# B&R Automation Studio project Kontrol
Automation Studio 4.9

## Configuration Config1

CPU X20CP1382, AutomationRuntime D4.83, Build 4.1.2

### Task classes (Cpu.sw)
```
Cyclic#1 (cycle 2000 us, tolerance 2000 us):
  TaskFast <- Kontrol.TaskFast.TaskFast.prg
  FastMeter <- (binary)
  Program <- (binary)
  SslClient <- (binary)
  Server <- (binary)
  Client <- (binary)
  TEXC <- (binary)
  Modbus <- (binary)
Cyclic#2 (cycle 10000 us, tolerance 10000 us):
  Protection <- Kontrol.Protection.Protection.prg
  Control <- Kontrol.Control.Control.prg
Cyclic#3 (cycle 100000 us, tolerance 100000 us):
  WatchDog <- WatchDog.WatchDog.prg
  System <- Kontrol.System.System.prg
  Hardware <- Kontrol.Hardware.Hardware.prg
  ProtUpdate <- Kontrol.Protection.ProtUpdate.prg
  Command <- Kontrol.Command.Command.prg
  cb52 <- Kontrol.CB52.cb52.prg
Cyclic#4 (cycle 200000 us, tolerance 200000 us):
  Auto <- Auto.Auto.prg
  RV <- (binary)
  UHLM <- (binary)
  UHLM_AL <- (binary)
  Alarme <- (binary)
  DJ52G_IO <- (binary)
  Comandos <- (binary)
  RT <- (binary)
  SFA_IO <- (binary)
  FREIO <- (binary)
  UHRV_IO <- (binary)
  Comp_IO <- (binary)
  SC <- (binary)
  Comp_UH_AL <- (binary)
  Turbina_IO <- (binary)
  DJ52G <- (binary)
  UHRV <- (binary)
  SA <- (binary)
  Comp_UH_IO <- (binary)
  Gerador_AL <- (binary)
  Turbina_AL <- (binary)
  Comp_UH <- (binary)
  UHRV_AL <- (binary)
  Partida <- (binary)
  SFA <- (binary)
  UHLM_IO <- (binary)
  Gerador_IO <- (binary)
  Parada <- (binary)
  Status <- (binary)
  Comp <- (binary)
  Painel <- (binary)
  Energia <- (binary)
  FA <- (binary)
  Comp_AL <- (binary)
  SFA_AL <- (binary)
Cyclic#5 (cycle 500000 us, tolerance 500000 us):
  Nivel_IO <- (binary)
  Nivel <- (binary)
Cyclic#6 (cycle 100000 us, tolerance 3000000 us):
  MDB_Comand <- Auto.Modbus.MDB_Comando.prg
  MDB_Status <- Auto.Modbus.MDB_Status.prg
  MDB_Alarme <- Auto.Modbus.MDB_Alarme.prg
  MDB_Medida <- Auto.Modbus.MDB_Medida.prg
  MDB_Parame <- Auto.Modbus.MDB_Parametro.prg
Cyclic#7 (cycle 20000 us, tolerance 10000000 us):
  Event <- Kontrol.Event.Event.prg
  Comm <- Comm.Comm.prg
Cyclic#8 (cycle 50000 us, tolerance 10000000 us):
  File <- Kontrol.File.File.prg
Binaries: TCData, udbdef, ashwd, sysconf, asfw, arconfig, iomap, Role, User, ashwac, OpcUaMap, vccddbox, ihm01, ihm02, ihm03, vccpopup, vcpfx20, vcctrend, vccstr, vcmgr, vcpdsw, vcpdvnc, vccline, vccovl, arial, vcdsint, vccnum, vcalarm, vctcal, vccbtn, vcnet, vccbmp, vcrt, vcshared, vccdt, vcgclass, vcfntttf, vcbclass, vcdsloc, vcfile, arialbd, vcctext, vccshape, vccgauge, vcpkat, 10111548$f, Visu02, Visu03, Visu01, vccbar, vccslider, vcchspot, vccurl, vccalarm, vcchtml, vcxml
Libraries: operator, runtime, LoopConR, sys_lib, brsystem, AsTCP, AsIecCon, astime, AsBrStr, AsARCfg, AsXml, FileIO, AsIOAcc, standard, AsSem, IecCheck, DRV_mbus, dvframe, DataObj, Pgs0985, PgsAI4622, PgsAO4622, PgsAuto, PgsCfgNet, PgsComm, PgsControl, PgsEvent, PgsFileSys, PgsProt, PgsTag, PgsTagLink, PgsTelnet, vcresman, ashw
```

### Hardware
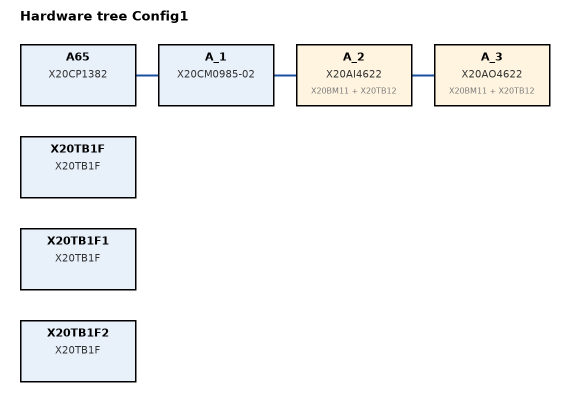
```
A65 : X20CP1382 v1.8.0.0  [X1 -> X1.SL; X2 -> X2.SL; X3 -> X3.SL]
  Module X1 (Type=X1, Virtual=true, Version=1.8.0.0)
    Connection (Connector=SS1, TargetModule=X20TB1F, TargetConnector=SS)
    Connection (Connector=SL, TargetModule=A65, TargetConnector=X1)
    X1AI_ChannelType01 = PT1000
    X1AI_ChannelType02 = 4 to 20mA
    X1AI2_LowerLimit_420mA = -8192
  Module X2 (Type=X2, Virtual=true, Version=1.8.0.0)
    Connection (Connector=SS1, TargetModule=X20TB1F1, TargetConnector=SS)
    Connection (Connector=SL, TargetModule=A65, TargetConnector=X2)
    X2CounterFunction = Edge
    X2CounterTimeInfo = 32Bit
  Module X3 (Type=X3, Virtual=true, Version=1.8.0.0)
    Connection (Connector=SS1, TargetModule=X20TB1F2, TargetConnector=SS)
    Connection (Connector=SL, TargetModule=A65, TargetConnector=X3)
  Connector IF2:
    ActivateDevice = 1
    HostName = kontrol
    Mode = Manual
    InternetAddress = 10.201.3.9
    SubnetMask = 255.255.255.192
    InaNodeNumber = 6
    Vnc1
    VncKeyMappingFile1 = 
    VncRefreshRate1 = 250
    ActivateSnmp = 2
    ActivateModbus = 1
    NumSlaves = -1
    NumAllBlocks = -1
    MemSizeIn = -1
    MemSizeOut = -1
  Connector IF3:
    CycleTime = 2000
    EPL_LossFrameTolerance_Selector = 2
    EPL_LossFrameTolerance = 5
    ActivateIna = 1
    InaNodeNumber = 1
  ConfigurationID = A65
  RemanentGlobalPvSize = 10940
  EnableUsbRemoteInstall = 1
  EnableCfRemoteInstall = 1
  SystemTick = 1000
  IdleTaskClass = 8
  TaskClassIdleTime = 4000
  Cyclic1Duration = 2000
  Cyclic1Tolerance = 2000
  Cyclic2Duration = 10000
  Cyclic2Tolerance = 10000
  Cyclic3Duration = 100000
  Cyclic3Tolerance = 100000
  Cyclic4Duration = 200000
  Cyclic4Tolerance = 200000
  Cyclic5Duration = 500000
  Cyclic5Tolerance = 500000
  Cyclic6Duration = 100000
  Cyclic6Tolerance = 3000000
  Cyclic7Duration = 20000
  Cyclic7Tolerance = 10000000
  Cyclic8Duration = 50000
  Cyclic8Tolerance = 10000000
  FileDevice1
  FileDeviceName1 = 
  FileDevicePath1 = 
  TimeZone = 105
  ActivateSntp = 1
  SntpcServAddr1 = a.st1.ntp.br
  SntpcServAddr2 = b.st1.ntp.br
  SntpcServAddr3 = c.st1.ntp.br
  SntpcServAddr4 = d.st1.ntp.br
  EthernetHostName = kontrol
  EthernetDefaultGateway = 10.201.3.62
  FtpUser1
  FtpUsername1 = progressul
  FtpUserPassword1 = vk2iY3J4UkERtYbEJrmZIzULlFJLyE0YoKo7iPp2s1I=
  FtpUserSalt1 = 6vig95Eg
  FTPAccessRight1 = 0
  FTPMSPartition1 = SYSTEM
  FTPMSpath1 = 
  ActivateOpcUa = 1
  OpcUaInformationModels_PV_Version = 1
A_1 : X20CM0985-02 v1.3.0.0  [X2X1 -> A65.IF6]
  Supervision = off
  ReadBack = on
  FuncDO5 = NetErrorUser
  Timestamps = on
  GenErrorReset = on
  GenErrorCheck = phaseline
  NetConfig = 3Phase
  SyncConfig = X4X3
A_2 : X20AI4622 v1.0.5.0  [SS1 -> X20TB12e.SS; SL -> X20BM11e.SL1]
  Supervision = off
  ChannelType01 = 4 to 20mA
  ChannelType02 = 4 to 20mA
  ChannelType03 = 4 to 20mA
  ChannelType04 = 4 to 20mA
A_3 : X20AO4622 v1.3.0.0  [SS1 -> X20TB12j.SS; SL -> X20BM11i.SL1]
  Supervision = off
  ChannelType01 = 0 to 20mA
  ChannelType02 = 4 to 20mA
  ChannelType03 = 4 to 20mA
  ChannelType04 = 4 to 20mA
X20BM11e : X20BM11 v1.0.0.1  [X2X1 -> A_1.X2X2]
X20BM11i : X20BM11 v1.0.0.1  [X2X1 -> X20BM11e.X2X2]
X20TB12e : X20TB12 v1.0.0.0
X20TB12j : X20TB12 v1.0.0.0
X20TB1F : X20TB1F v1.0.0.0
X20TB1F1 : X20TB1F v1.0.0.0
X20TB1F2 : X20TB1F v1.0.0.0
```

### IoMap.iom - A65/IoMap.iom
```iecst
(*********************************************************************************
 * Copyright: Microsoft
 * Author:    sandrionir
 * Created:   February 21, 2017/7:19 AM
 *********************************************************************************
 * IO mapping
 *********************************************************************************)
VAR_CONFIG
	Cyclic#2.::Control:rpm2.MasterCount AT %ID."X2".Counter02Value;
	Cyclic#2.::Control:rpm2.MasterTime AT %ID."X2".Counter02TimeChanged;
	Cyclic#2.::Control:rpm1.MasterCount AT %ID."X2".Counter01Value;
	Cyclic#2.::Control:rpm1.MasterTime AT %ID."X2".Counter01TimeChanged;
	Cyclic#2.cm0985IO.di.T32N AT %IX."A_1".StatusInput32;
	Cyclic#2.cm0985IO.di.T32P AT %IX."A_1".StatusInput31;
	Cyclic#2.cm0985IO.di.T27_2 AT %IX."A_1".StatusInput18;
	Cyclic#2.cm0985IO.di.T32Q AT %IX."A_1".StatusInput10;
	Cyclic#2.cm0985IO.di.T51 AT %IX."A_1".StatusInput09;
	Cyclic#2.cm0985IO.di.T50 AT %IX."A_1".StatusInput08;
	Cyclic#2.cm0985IO.di.T50N AT %IX."A_1".StatusInput07;
	Cyclic#2.cm0985IO.di.T60I AT %IX."A_1".StatusInput06;
	Cyclic#2.cm0985IO.di.T60V AT %IX."A_1".StatusInput05;
	Cyclic#2.cm0985IO.di.T81U AT %IX."A_1".StatusInput04;
	Cyclic#2.cm0985IO.di.T81O AT %IX."A_1".StatusInput03;
	Cyclic#2.cm0985IO.di.T27_1 AT %IX."A_1".StatusInput02;
	Cyclic#2.cm0985IO.di.T59 AT %IX."A_1".StatusInput01;
	Cyclic#2.cm0985IO.di.UgPhSeqFault AT %IX."A_1".StatusInput19;
	Cyclic#2.cm0985IO.di.IgPhSeqFault AT %IX."A_1".StatusInput20;
	Cyclic#2.cm0985IO.di.UbPhSeqFault AT %IX."A_1".StatusInput21;
	Cyclic#2.cm0985IO.di.Us1PhSeqFault AT %IX."A_1".StatusInput22;
	Cyclic#2.cm0985IO.di.PS24VFault AT %IX."A_1".StatusInput16;
	Cyclic#2.cm0985IO.do.RstError AT %QX."A_1".ResetGeneratorErrors;
	Cyclic#2.cm0985IO.do.INVDO05 AT %QX."A_1".InvertDO5;
	Cyclic#2.cm0985IO.do.SyncDeadBus AT %QX."A_1".ConfigOutput19;
	Cyclic#2.cm0985IO.do.SyncCheck AT %QX."A_1".ConfigOutput18;
	Cyclic#2.cm0985IO.do.SyncSlip AT %QX."A_1".ConfigOutput17;
	Cyclic#2.cm0985Meter.Registers.AnalogInput43 AT %ID."A_1".AnalogInput43;
	Cyclic#2.cm0985Meter.Registers.AnalogInput42 AT %ID."A_1".AnalogInput42;
	Cyclic#2.cm0985Meter.Registers.AnalogInput41 AT %ID."A_1".AnalogInput41;
	Cyclic#2.cm0985Meter.Registers.AnalogInput40 AT %ID."A_1".AnalogInput40;
	Cyclic#2.cm0985Meter.Registers.AnalogInput39 AT %ID."A_1".AnalogInput39;
	Cyclic#2.cm0985Meter.Registers.AnalogInput38 AT %ID."A_1".AnalogInput38;
	Cyclic#2.cm0985Meter.Registers.AnalogInput35 AT %IW."A_1".AnalogInput35;
	Cyclic#2.cm0985Meter.Registers.AnalogInput30 AT %IW."A_1".AnalogInput30;
	Cyclic#2.cm0985Meter.Registers.AnalogInput29 AT %IW."A_1".AnalogInput29;
	Cyclic#2.cm0985Meter.Registers.AnalogInput27 AT %IW."A_1".AnalogInput27;
	Cyclic#2.cm0985Meter.Registers.AnalogInput26 AT %IW."A_1".AnalogInput26;
	Cyclic#2.cm0985Meter.Registers.AnalogInput25 AT %IW."A_1".AnalogInput25;
	Cyclic#2.cm0985Meter.Registers.AnalogInput24 AT %IW."A_1".AnalogInput24;
	Cyclic#2.cm0985Meter.Registers.AnalogInput23 AT %IW."A_1".AnalogInput23;
	Cyclic#2.cm0985Meter.Registers.AnalogInput22 AT %IW."A_1".AnalogInput22;
	Cyclic#2.cm0985Meter.Registers.AnalogInput21 AT %IW."A_1".AnalogInput21;
	Cyclic#2.cm0985Meter.Registers.AnalogInput20 AT %IW."A_1".AnalogInput20;
	Cyclic#2.cm0985Meter.Registers.AnalogInput19 AT %IW."A_1".AnalogInput19;
	Cyclic#2.cm0985Meter.Registers.AnalogInput18 AT %IW."A_1".AnalogInput18;
	Cyclic#2.cm0985Meter.Registers.AnalogInput17 AT %IW."A_1".AnalogInput17;
	Cyclic#2.cm0985Meter.Registers.AnalogInput16 AT %IW."A_1".AnalogInput16;
	Cyclic#2.cm0985Meter.Registers.AnalogInput15 AT %IW."A_1".AnalogInput15;
	Cyclic#2.cm0985Meter.Registers.AnalogInput14 AT %IW."A_1".AnalogInput14;
	Cyclic#2.cm0985Meter.Registers.AnalogInput13 AT %IW."A_1".AnalogInput13;
	Cyclic#2.cm0985Meter.Registers.AnalogInput12 AT %IW."A_1".AnalogInput12;
	Cyclic#2.cm0985Meter.Registers.AnalogInput11 AT %IW."A_1".AnalogInput11;
	Cyclic#2.cm0985Meter.Registers.AnalogInput10 AT %IW."A_1".AnalogInput10;
	Cyclic#2.cm0985Meter.Registers.AnalogInput09 AT %IW."A_1".AnalogInput09;
	Cyclic#2.cm0985Meter.Registers.AnalogInput08 AT %IW."A_1".AnalogInput08;
	Cyclic#2.cm0985Meter.Registers.AnalogInput07 AT %IW."A_1".AnalogInput07;
	Cyclic#2.cm0985Meter.Registers.AnalogInput06 AT %IW."A_1".AnalogInput06;
	Cyclic#2.cm0985Meter.Registers.AnalogInput05 AT %IW."A_1".AnalogInput05;
	Cyclic#2.cm0985Meter.Registers.AnalogInput04 AT %IW."A_1".AnalogInput04;
	Cyclic#2.cm0985Meter.Registers.AnalogInput03 AT %IW."A_1".AnalogInput03;
	Cyclic#2.cm0985Meter.Registers.AnalogInput02 AT %IW."A_1".AnalogInput02;
	Cyclic#2.cm0985Meter.Registers.AnalogInput01 AT %IW."A_1".AnalogInput01;
	Cyclic#2.cm0985Meter.Registers.AnalogInput33 AT %IW."A_1".AnalogInput33;
	Cyclic#2.cm0985Meter.Registers.AnalogInput34 AT %IW."A_1".AnalogInput34;
	Cyclic#2.cm0985Meter.Registers.AnalogInput31 AT %IW."A_1".AnalogInput31;
	Cyclic#2.cm0985Meter.Registers.AnalogInput32 AT %IW."A_1".AnalogInput32;
	HW.SerialNumber AT %ID."A65".SerialNumber;
	HW.ModuleID AT %IW."A65".ModuleID;
	HW.TemperatureENV AT %IW."A65".TemperatureENV;
	HW.TemperatureCPU AT %IW."A65".TemperatureCPU;
	HW.FalhaFonteIO AT %IX."X3".StatusInput01;
	HW.Modulos.X1_Status AT %IB."X1".StatusInput01;
	HW.Modulos.A_1_OK AT %IX."A_1".ModuleOk;
	HW.Modulos.A_2_OK AT %IX."A_2".ModuleOk;
	HW.Modulos.A_3_OK AT %IX."A_3".ModuleOk;
	Protection.ai.ExcTemp AT %IW."X1".AnalogInput01;
	A65.ai.if AT %IW."X1".AnalogInput02;
	A65.ai.uf AT %IW."A_2".AnalogInput01;
	A65.ai.pos1 AT %IW."A_2".AnalogInput02;
	A65.ai.pos2 AT %IW."A_2".AnalogInput03;
	A65.ai.pos3 AT %IW."A_2".AnalogInput04;
	A65.ao.pwr AT %QW."A_3".AnalogOutput01;
	A65.ao.pos1 AT %QW."A_3".AnalogOutput02;
	A65.ao.pos2 AT %QW."A_3".AnalogOutput03;
	A65.ao.pos3 AT %QW."A_3".AnalogOutput04;
	A65.di.reset  AT %IX."X1".DigitalInput01;
	A65.di.gov_enable  AT %IX."X1".DigitalInput02;
	A65.di.gov_ctrl_pwr_enable AT %IX."X1".DigitalInput03;
	A65.di.gov_unload AT %IX."X1".DigitalInput04;
	A65.di.avr_enable AT %IX."X2".DigitalInput01;
	A65.di.avr_ctrl_qm_enable AT %IX."X2".DigitalInput02;
	A65.di.avr_ctrl_pf_enable AT %IX."X2".DigitalInput03;
	A65.di.sync_enable AT %IX."X2".DigitalInput04;
	A65.di.dead_bus_enable AT %IX."X2".DigitalInput05;
	A65.di.remote AT %IX."X2".DigitalInput07;
	A65.di.gov_trip AT %IX."X2".DigitalInput08;
	A65.di.avr_trip AT %IX."X2".DigitalInput09;
	CB52.di.closed AT %IX."X2".DigitalInput06;
	Protection.di.crowbar_ok AT %IX."X2".DigitalInput10;
	Protection.di.pwr_temp_ok AT %IX."X2".DigitalInput14;
	Protection.do.trip_86e AT %QX."A_1".DigitalOutput05;
	Protection.do.trip_86h AT %QX."A_1".DigitalOutput06;
	Protection.do.trip_50bf AT %QX."X3".DigitalOutput12;
	A65.do.gov_on AT %QX."X3".DigitalOutput02;
	A65.do.watchdog AT %QX."X3".DigitalOutput01;
	A65.do.power_zero AT %QX."X3".DigitalOutput03;
	A65.do.rotation_zero AT %QX."X3".DigitalOutput04;
	A65.do.rotation_nominal AT %QX."X3".DigitalOutput05;
	A65.do.rotation_brake AT %QX."X3".DigitalOutput06;
	A65.do.avr_on AT %QX."X3".DigitalOutput07;
	A65.do.field_flash_on AT %QX."X3".DigitalOutput08;
	A65.do.voltage_nominal AT %QX."X3".DigitalOutput09;
	A65.do.sync_enabled AT %QX."X3".DigitalOutput10;
	A65.do.dead_bus_enabled AT %QX."X3".DigitalOutput11;
END_VAR
```

## Logical view

Binary libraries used (declarations not repeated): operator, runtime, LoopConR 4.10.0, sys_lib, brsystem, AsTCP, AsIecCon, astime, AsARCfg, FileIO, standard, AsSem, AsIOAcc, AsXml, AsBrStr, DRV_mbus, dvframe, DataObj, IecCheck, Pgs0985, PgsAI4622 1.00.0, PgsAO4622 1.00.0, PgsCfgNet 2.02.0, PgsComm, PgsControl 2.03.3, PgsEvent, PgsFileSys 2.00.0, PgsTag, PgsTagLink 2.00.0, PgsTelnet

### Package Logical/Libraries - Global libraries

### Library Logical/Libraries/Kontrol/PgsAuto (IEC)
Depends on: sys_lib

#### Types.typ - Exported data types
```iecst
TYPE
	PgsHorimetroPrivType : 	STRUCT
		init : BOOL := TRUE;
		init_ton : TON;
		sec_old : USINT;
		rtc_time : RTCtime_typ;
		bkp_ton : TON;
	END_STRUCT;
	PgsManobraPrivType : 	STRUCT
		init : BOOL := TRUE;
		init_ton : TON;
		bkp_ton : TON;
		m : BOOL;
	END_STRUCT;
	PgsEnergiaPrivType : 	STRUCT
		init : BOOL := TRUE;
		init_ton : TON;
		dh : REAL; (*Delta Hour*)
		rt_info : RTInfo;
		bkp_ton : TON;
	END_STRUCT;
END_TYPE
```

#### PgsAuto.fun - Exported functions and function blocks
```iecst
FUNCTION_BLOCK PgsEnergia
	VAR_INPUT
		enable : BOOL;
		reset : BOOL;
		power : REAL;
		set_inicial : BOOL;
		set_posEnergy : REAL;
		set_negEnergy : REAL;
	END_VAR
	VAR_OUTPUT
		posEnergy : LREAL;
		negEnergy : LREAL;
	END_VAR
	VAR
		priv : PgsEnergiaPrivType;
	END_VAR
END_FUNCTION_BLOCK

FUNCTION_BLOCK PgsHorimetro
	VAR_INPUT
		enable : BOOL;
		reset : BOOL;
		set_inicial : BOOL;
		set_total : REAL;
	END_VAR
	VAR_OUTPUT
		total : REAL;
		horas : REAL;
		minutos : REAL;
		segundos : REAL;
	END_VAR
	VAR
		priv : PgsHorimetroPrivType;
	END_VAR
END_FUNCTION_BLOCK

FUNCTION_BLOCK PgsManobra
	VAR_INPUT
		enable : BOOL;
		reset : BOOL;
		set_inicial : BOOL;
		set_total : REAL;
	END_VAR
	VAR_OUTPUT
		total : REAL;
	END_VAR
	VAR
		priv : PgsManobraPrivType;
	END_VAR
END_FUNCTION_BLOCK

FUNCTION PGS_MDB_TO_REAL : REAL (*TODO: Add your comment here*) (*$GROUP=User,$CAT=User,$GROUPICON=User.png,$CATICON=User.png*)
	VAR_INPUT
		IN : UDINT;
	END_VAR
	VAR
		pVar : REFERENCE TO REAL;
		varUint : ARRAY[0..1] OF UINT;
		varUint1 : REFERENCE TO ARRAY[0..1] OF UINT;
	END_VAR
END_FUNCTION

FUNCTION PGS_REAL_TO_MDB : UDINT (*TODO: Add your comment here*) (*$GROUP=User,$CAT=User,$GROUPICON=User.png,$CATICON=User.png*)
	VAR_INPUT
		IN : REAL;
	END_VAR
	VAR
		pVar : REFERENCE TO UDINT;
		varUint : ARRAY[0..1] OF UINT;
		varUint1 : REFERENCE TO ARRAY[0..1] OF UINT;
	END_VAR
END_FUNCTION

{REDUND_ERROR} FUNCTION PGS_MDB_TO_DINT : DINT (*TODO: Add your comment here*) (*$GROUP=User,$CAT=User,$GROUPICON=User.png,$CATICON=User.png*)
	VAR_INPUT
		HIGH : UINT;
		LOW : UINT;
	END_VAR
	VAR
		pVar : REFERENCE TO DINT;
		varUint : ARRAY[0..1] OF UINT;
	END_VAR
END_FUNCTION

{REDUND_ERROR} FUNCTION PGS_MDB_TO_UDINT : UDINT (*TODO: Add your comment here*) (*$GROUP=User,$CAT=User,$GROUPICON=User.png,$CATICON=User.png*)
	VAR_INPUT
		HIGH : UINT;
		LOW : UINT;
	END_VAR
	VAR
		pVar : REFERENCE TO UDINT;
		varUint : ARRAY[0..1] OF UINT;
	END_VAR
END_FUNCTION

FUNCTION_BLOCK PgsAlarme
	VAR_INPUT
		IN : BOOL; (*input signal*)
		PT : TIME; (*delay time*)
		RESET : BOOL; (*resets output Q1*)
	END_VAR
	VAR_OUTPUT
		Q : BOOL; (*rising edge of the input signal is delayed by PT*)
	END_VAR
	VAR
		ton : TON;
	END_VAR
END_FUNCTION_BLOCK

{REDUND_ERROR} FUNCTION_BLOCK PgsFiltro (*TODO: Add your comment here*) (*$GROUP=User,$CAT=User,$GROUPICON=User.png,$CATICON=User.png*)
	VAR_INPUT
		IN : {REDUND_UNREPLICABLE} REAL;
		CTE : {REDUND_UNREPLICABLE} REAL;
	END_VAR
	VAR_OUTPUT
		OUT : {REDUND_UNREPLICABLE} REAL;
	END_VAR
	VAR
		acc : REAL;
	END_VAR
END_FUNCTION_BLOCK

{REDUND_ERROR} FUNCTION_BLOCK PgsEscala (*TODO: Add your comment here*) (*$GROUP=User,$CAT=User,$GROUPICON=User.png,$CATICON=User.png*)
	VAR_INPUT
		SensorMax : {REDUND_UNREPLICABLE} REAL;
		SensorMin : {REDUND_UNREPLICABLE} REAL;
		Filtro : REAL;
		Entrada : REAL;
	END_VAR
	VAR_OUTPUT
		Valor : {REDUND_UNREPLICABLE} REAL;
		Sensor : REAL;
	END_VAR
	VAR
		priv_filtro : PgsFiltro;
		priv_first_start : BOOL;
	END_VAR
END_FUNCTION_BLOCK

{REDUND_ERROR} FUNCTION_BLOCK PgsCabo (*TODO: Add your comment here*) (*$GROUP=User,$CAT=User,$GROUPICON=User.png,$CATICON=User.png*)
	VAR_INPUT
		IN : REAL;
		PT : TIME;
	END_VAR
	VAR_OUTPUT
		Falha : BOOL;
		Cabo_Aberto : BOOL;
		Cabo_Curto : BOOL;
	END_VAR
	VAR
		aberto : BOOL;
		curto : BOOL;
		ton_aberto : TON;
		ton_curto : TON;
	END_VAR
END_FUNCTION_BLOCK

{REDUND_OK} FUNCTION_BLOCK PgsSobre (*TODO: Add your comment here*) (*$GROUP=User,$CAT=User,$GROUPICON=User.png,$CATICON=User.png*)
	VAR_INPUT
		enable : BOOL := TRUE;
		IN : REAL;
		IN_AL : REAL;
		PT_AL : REAL;
		IN_TP : REAL;
		PT_TP : REAL;
		RST : BOOL;
	END_VAR
	VAR_OUTPUT
		Alarme : BOOL;
		Trip : BOOL;
	END_VAR
	VAR
		ton_al : TON;
		ton_tp : TON;
	END_VAR
END_FUNCTION_BLOCK

{REDUND_OK} FUNCTION_BLOCK PgsSub (*TODO: Add your comment here*) (*$GROUP=User,$CAT=User,$GROUPICON=User.png,$CATICON=User.png*)
	VAR_INPUT
		enable : BOOL := TRUE;
		IN : REAL;
		IN_AL : REAL;
		PT_AL : REAL;
		IN_TP : REAL;
		PT_TP : REAL;
		RST : BOOL;
	END_VAR
	VAR_OUTPUT
		Alarme : BOOL;
		Trip : BOOL;
	END_VAR
	VAR
		ton_al : TON;
		ton_tp : TON;
	END_VAR
END_FUNCTION_BLOCK

FUNCTION_BLOCK PgsX20AT
	VAR_INPUT
		Status : USINT;
	END_VAR
	VAR_OUTPUT
		IN1_Aberto : BOOL;
		IN1_Curto : BOOL;
		IN2_Aberto : BOOL;
		IN2_Curto : BOOL;
		IN3_Aberto : BOOL;
		IN3_Curto : BOOL;
		IN4_Aberto : BOOL;
		IN4_Curto : BOOL;
	END_VAR
END_FUNCTION_BLOCK

{REDUND_ERROR} FUNCTION_BLOCK PgsEscalaTotal (*TODO: Add your comment here*) (*$GROUP=User,$CAT=User,$GROUPICON=User.png,$CATICON=User.png*)
	VAR_INPUT
		SensorMax : {REDUND_UNREPLICABLE} REAL;
		SensorMin : {REDUND_UNREPLICABLE} REAL;
		ValorMax : {REDUND_UNREPLICABLE} REAL;
		ValorMin : {REDUND_UNREPLICABLE} REAL;
		Entrada : REAL;
	END_VAR
	VAR_OUTPUT
		Valor : {REDUND_UNREPLICABLE} REAL;
		Sensor : REAL;
	END_VAR
END_FUNCTION_BLOCK
```

#### PgsHorimetro.st
```iecst
FUNCTION_BLOCK PgsHorimetro

	priv.init_ton(IN:= priv.init, PT:=T#10s);
	IF priv.init_ton.Q THEN
		priv.init := FALSE;
		total := set_total;
	END_IF;

	RTC_gettime(ADR(priv.rtc_time));
	IF reset THEN
		reset 	:= FALSE;
		total 	:= 0.0;
	END_IF;

	IF enable AND priv.sec_old <> priv.rtc_time.second THEN
		total := total + 1.0 / 3600.0;
	END_IF;
	priv.sec_old := priv.rtc_time.second;

	IF set_inicial THEN
		set_inicial := FALSE;
		total := set_total;
	END_IF;

	horas	:= TRUNC(total);
	minutos	:= TRUNC((total - horas)*60.0);
	segundos:= TRUNC((total - horas - minutos/60.0)*3600.0);

	priv.bkp_ton(IN:= NOT priv.bkp_ton.Q, PT:=T#10m);
	IF priv.bkp_ton.Q THEN
		set_total := total;
	END_IF;
END_FUNCTION_BLOCK
```

#### PgsManobra.st
```iecst
FUNCTION_BLOCK PgsManobra
	priv.init_ton(IN:= priv.init, PT:=T#10s);
	IF priv.init_ton.Q THEN
		priv.init := FALSE;
		total := set_total;
	END_IF;

    IF reset THEN
    	reset	:= FALSE;
        total	:= 0;
    END_IF;

	IF set_inicial THEN
		set_inicial	:= FALSE;
		total	:= set_total;
	END_IF;

    IF NOT priv.m AND enable THEN total := total + 1.0; END_IF;
    priv.m := enable;

	priv.bkp_ton(IN:= NOT priv.bkp_ton.Q, PT:=T#1m);
	IF priv.bkp_ton.Q THEN
		set_total := total;
	END_IF;
END_FUNCTION_BLOCK
```

#### PGS_MDB_TO_UDINT.st
```iecst
(* TODO: Add your comment here *)
FUNCTION PGS_MDB_TO_UDINT
    varUint[0] := HIGH;
    varUint[1] := LOW;
    pVar ACCESS ADR(varUint);
    PGS_MDB_TO_UDINT := pVar;
END_FUNCTION
```

#### PgsCabo.st
```iecst
(* TODO: Add your comment here *)
FUNCTION_BLOCK PgsCabo
	curto 	:= IN >= 20.0;
	aberto	:= IN <= 3.0;
	ton_aberto(IN:=aberto,PT:=PT);
	ton_curto(IN:=curto,PT:=PT);
	Falha 		:= aberto OR curto;
	Cabo_Aberto	:= ton_aberto.Q;
	Cabo_Curto	:= ton_curto.Q;
END_FUNCTION_BLOCK
```

#### PgsSub.st
```iecst
(*<$Description$> TODO: Add your comment here </$Description$>*)
FUNCTION_BLOCK PgsSub

	(* Alarme *)
	IF IN_AL = 0 THEN
		Alarme	:= FALSE;
	ELSE
		ton_al( IN := IN <= IN_AL , PT := REAL_TO_TIME( PT_AL * 1000) );
		IF ton_al.Q AND enable THEN
			Alarme	:= TRUE;
		ELSIF RST THEN
			Alarme	:= FALSE;
		END_IF;
	END_IF;

	(*Trip*)
	IF IN_TP = 0 THEN
		Trip	:= FALSE;
	ELSE
		ton_tp( IN := IN <= IN_TP , PT := REAL_TO_TIME( PT_TP * 1000) );
		IF ton_tp.Q AND enable THEN
			Trip	:= TRUE;
		ELSIF RST THEN
			Trip	:= FALSE;
		END_IF;
 	END_IF;

END_FUNCTION_BLOCK
```

#### PgsX20AT.st
```iecst
(*<$Description$> TODO: Add your comment here </$Description$>*)
FUNCTION_BLOCK PgsX20AT
	IN1_Aberto		:= Status.0;
	IN1_Curto		:= (Status.1 = 1) AND (Status.0 = 0);

	IN2_Aberto		:= Status.2;
	IN2_Curto		:= (Status.3 = 1) AND (Status.2 = 0);

	IN3_Aberto		:= Status.4;
	IN3_Curto		:= (Status.5 = 1) AND (Status.4 = 0);

	IN4_Aberto		:= Status.6;
	IN4_Curto		:= (Status.7 = 1) AND (Status.6 = 0);

END_FUNCTION_BLOCK
```

#### PgsEscalaTotal.st
```iecst
(* TODO: Add your comment here *)
FUNCTION_BLOCK PgsEscalaTotal

	Sensor	:= (Entrada / 32767.0) * 16.0 + 4.0;
	IF (SensorMax - SensorMin) <> 0 THEN
		Valor   := ((Sensor - SensorMin) / (SensorMax - SensorMin))
				* (ValorMax - ValorMin)
				+  ValorMin;
	ELSE
		Valor   := 0.0;
	END_IF;

END_FUNCTION_BLOCK
```

#### PgsEscala.st
```iecst
(* TODO: Add your comment here *)
FUNCTION_BLOCK PgsEscala

	Sensor	:= (Entrada / 32767.0) * 16.0 + 4.0;

	IF Filtro < 1 THEN
		Filtro := 1;
	END_IF
	priv_filtro(IN:=Sensor, CTE:=Filtro);

	IF NOT priv_first_start THEN
		priv_first_start := TRUE;
		priv_filtro(IN:= (Sensor - (priv_filtro.acc / Filtro) ) * Filtro);
	END_IF;

	Valor   := ((priv_filtro.OUT - 4.0) / 16.0)
	* (SensorMax - SensorMin)
	+  SensorMin;

END_FUNCTION_BLOCK
```

### Share.var
```iecst
VAR
	WDOK : BOOL := TRUE;
	License : PgsLicense;
END_VAR
```

### Program Logical/WatchDog/WatchDog

#### Cyclic.st
```iecst
PROGRAM _CYCLIC
    License();
    ProtFlag.KeyInvalid			:= NOT License.Valid;
    ProtFlag.PwrSrcCpuIOFault	:= HW.FalhaFonteIO;
    ProtFlag.PwrSrcM1IOFault	:= cm0985IO.di.PS24VFault;

    IF  License.Valid
    AND	NOT ProtFlag.PwrSrcCpuIOFault	// Power Source CPU I/O Fault
    AND	NOT ProtFlag.PwrSrcM1IOFault	// Power Source Energy Module I/O Fault
    AND	HW.Modulos.A_1_OK
    AND	HW.Modulos.A_2_OK
	AND	HW.Modulos.A_3_OK
//	AND	HW.Modulos.A_4_OK
//	AND	HW.Modulos.A_5_OK
//	AND	HW.Modulos.A_6_OK
//	AND	HW.Modulos.A_7_OK
//	AND	HW.Modulos.A_8_OK
//	AND	HW.Modulos.A_9_OK
//	AND	HW.Modulos.A_10_OK
//	AND	HW.Modulos.A_11_OK
//	AND	HW.Modulos.A_12_OK
	THEN
        WDOK    := TRUE;
    ELSE
        WDOK    := FALSE;
    END_IF

    //WatchDog
    ProtFlag.WatchDog	:= NOT WDOK;
	A65.do.watchdog		:= WDOK;

END_PROGRAM
```

- Cyclic.st.bak (not shown)

### Program Logical/Comm/Comm (IEC)

#### Variables.var
```iecst
VAR
	mbusData : PgsMbDataOpen;
	mbusDevice : PgsMbDevice;
	mbusSetBlock : PgsMbSetBlock;
	mbusSetLink : PgsMbSetLink;
	mbusDataClose : PgsMbDataClose;
	mbusLinkClose : PgsMbLinkClose;
	mbusTcpOpen : PgsMbTcpOpen;
	mbusTcpUpdate : PgsMbTcpUpdate;
	mbusTcpClose : PgsMbTcpClose;
	telnetOpen : PgsTelnetOpen;
	telnetUpdate : PgsTelnetUpdate;
	telnetClose : PgsTelnetClose;
END_VAR
(*Reset COM*)
VAR
	ton_reset_Tcp : TON;
END_VAR
```

#### Cyclic.st
```iecst
PROGRAM _CYCLIC

    IF NOT PgsTagValid(TagManager.ident) THEN
        RETURN;
    END_IF

    mbusTcpUpdate   ( ident := mbusTcpOpen.ident );
    telnetUpdate(
        ident       := telnetOpen.ident,
        tagIdent    := TagManager.ident,
        evtIdent    := Event
    );

	ton_reset_Tcp(IN:= A65.di.reset, PT:= T#30s);
	IF ton_reset_Tcp.Q THEN
		mbusTcpUpdate.reset := TRUE;
	END_IF;

END_PROGRAM
```

#### Exit.st
```iecst
PROGRAM _EXIT

	mbusDataClose( dtaIdent := mbusData.dtaIdent );

	mbusLinkClose( lnkIdent := link_avr.Ident );
	mbusLinkClose( lnkIdent := link_gov.Ident );

	mbusLinkClose( lnkIdent := link_pos1.Ident );
	mbusLinkClose( lnkIdent := link_pos2.Ident );
	mbusLinkClose( lnkIdent := link_pos3.Ident );
	mbusLinkClose( lnkIdent := link_curve1.Ident );
	mbusLinkClose( lnkIdent := link_curve2.Ident );
	mbusLinkClose( lnkIdent := link_curve3.Ident );

	mbusLinkClose( lnkIdent := link_meter.Ident );

	mbusLinkClose( lnkIdent := link_system.Ident );
	mbusLinkClose( lnkIdent := link_sysIO.Ident );
	mbusLinkClose( lnkIdent := link_prot.Ident );

    mbusTcpClose( enable := TRUE, ident := mbusTcpOpen.ident );

    telnetClose( enable := TRUE, ident := telnetOpen.ident );

END_PROGRAM
```

#### Init.st
```iecst
PROGRAM _INIT

    mbusData( Devices := 1 );

	//Device 1
    mbusDevice(
        dtaIdent        := mbusData.dtaIdent,
        id              := 1,
		Links			:= 6,
		InputBlocks		:= 1,
        CoilBlocks      := 3
    );

    //AVR
	link_avr(
		CoilAddress		:= 4097,
		HoldingAddress	:= 5121,
		InputAddress	:= 7169,
        //GainUm          := 10.0,
        //GainIm          := 10.0,
        //GainSm          := 10.0,
        //GainUf          := 100.0,
        //GainIf          := 100.0,
		Float			:= TRUE,
		ModiconFormat	:= TRUE
	);
	mbusSetLink(
		devIdent	:= mbusDevice.devIdent,
		lnkIdent	:= link_avr.Ident
	);

    //GOV
	link_gov(
		CoilAddress		:= 8193,
		HoldingAddress	:= 9217,
		InputAddress	:= 11265,
        //GainUm          := 10.0,
        //GainSm          := 10.0,
		Float			:= TRUE,
		ModiconFormat	:= TRUE
	);
	mbusSetLink(
		devIdent	:= mbusDevice.devIdent,
		lnkIdent	:= link_gov.Ident
	);

	//POS1
	link_pos1(
		CoilAddress		:= 12289,
		HoldingAddress	:= 12545,
		InputAddress	:= 13569,
		Float			:= TRUE,
		ModiconFormat	:= TRUE
	);
	mbusSetLink(
		devIdent	:= mbusDevice.devIdent,
		lnkIdent	:= link_pos1.Ident
	);
	//Curve1
	link_curve1(
		HoldingAddress	:= 13825,
		InputAddress	:= 13953,
		Float			:= TRUE,
		ModiconFormat	:= TRUE
	);
	mbusSetLink(
		devIdent	:= mbusDevice.devIdent,
		lnkIdent	:= link_curve1.Ident
	);

	//POS2
	link_pos2(
		CoilAddress		:= 14337,
		HoldingAddress	:= 14593,
		InputAddress	:= 15617,
		Float			:= TRUE,
		ModiconFormat	:= TRUE
	);
	mbusSetLink(
		devIdent	:= mbusDevice.devIdent,
		lnkIdent	:= link_pos2.Ident
	);
	//Curve2
	link_curve2(
		HoldingAddress	:= 15873,
		InputAddress	:= 16001,
		Float			:= TRUE,
		ModiconFormat	:= TRUE
	);
	mbusSetLink(
		devIdent	:= mbusDevice.devIdent,
		lnkIdent	:= link_curve2.Ident
	);

	//POS3
	link_pos3(
		CoilAddress		:= 16385,
		HoldingAddress	:= 16641,
		InputAddress	:= 17665,
		Float			:= TRUE,
		ModiconFormat	:= TRUE
	);
	mbusSetLink(
		devIdent	:= mbusDevice.devIdent,
		lnkIdent	:= link_pos3.Ident
	);
	//Curve3
	link_curve3(
		HoldingAddress	:= 17921,
		InputAddress	:= 18049,
		Float			:= TRUE,
		ModiconFormat	:= TRUE
	);
	mbusSetLink(
		devIdent	:= mbusDevice.devIdent,
		lnkIdent	:= link_curve3.Ident
	);

    // MdbMeter
	link_meter(
        pBlock	        := ADR(MdbMeter),
        blockLen	    := SIZEOF(MdbMeter),
		Address			:= 2561,
		Holding			:= FALSE,
		//Gain			:= 10.0,
		Float			:= TRUE,
		ModiconFormat	:= TRUE
	);
	mbusSetLink(
		devIdent	:= mbusDevice.devIdent,
		lnkIdent	:= link_meter.Ident
	);

    // System Parameter
	link_system(
        pBlock	        := ADR(SysPar),
        blockLen	    := SIZEOF(SysPar),
		Address			:= 1025,
		Holding			:= TRUE,
		//Gain			:= 10,
		Float			:= TRUE,
		ModiconFormat	:= TRUE
	);
	mbusSetLink(
		devIdent	:= mbusDevice.devIdent,
		lnkIdent	:= link_system.Ident
	);
    //
    link_sysIO(
        pBlock	        := ADR(SysIOPar),
        blockLen	    := SIZEOF(SysIOPar),
		Address			:= 1255,
		Holding			:= TRUE,
		//Gain			:= 10,
		Float			:= TRUE,
		ModiconFormat	:= TRUE
	);
	mbusSetLink(
		devIdent	:= mbusDevice.devIdent,
		lnkIdent	:= link_sysIO.Ident
	);

    //SysUpdate
 	mbusSetBlock(
        devIdent    := mbusDevice.devIdent,
        BlockType   := PGS_MB_BLK_COIL,
        Address     := 1,
        pBlock      := ADR(SysUpdate),
        blockLen    := SIZEOF(SysUpdate)
    );

    //Protections
 	mbusSetBlock(
        devIdent    := mbusDevice.devIdent,
        BlockType   := PGS_MB_BLK_COIL,
        Address     := 40961,
        pBlock      := ADR(ProtFlag),
        blockLen    := SIZEOF(ProtFlag)
	);
	// Protections Parameter
	link_prot(
		pBlock	        := ADR(ProtPar),
		blockLen	    := SIZEOF(ProtPar),
		Address			:= 41985,
		Holding			:= TRUE,
		//Gain			:= 10,
		Float			:= TRUE,
		ModiconFormat	:= TRUE
	);
	mbusSetLink(
		devIdent	:= mbusDevice.devIdent,
		lnkIdent	:= link_prot.Ident
	);

    //Automação
    link_mdb_medidas(
		pBlock	        := ADR(MDB_Medidas),
		blockLen	    := SIZEOF(MDB_Medidas),
		Address			:= 19089, (*50001*)
		Holding			:= FALSE,
		//Gain			:= 10,
		Float			:= TRUE,
		ModiconFormat	:= TRUE
	);
	mbusSetLink(
		devIdent	:= mbusDevice.devIdent,
		lnkIdent	:= link_mdb_medidas.Ident
	);
    link_mdb_parametros(
		pBlock	        := ADR(MDB_Parametros),
		blockLen	    := SIZEOF(MDB_Parametros),
		Address			:= 21589, (*50257*)
		Holding			:= TRUE,
		//Gain			:= 10,
		Float			:= TRUE,
		ModiconFormat	:= TRUE
	);
	mbusSetLink(
		devIdent	:= mbusDevice.devIdent,
		lnkIdent	:= link_mdb_parametros.Ident
	);
	mbusSetBlock(
		devIdent    := mbusDevice.devIdent,
		BlockType   := PGS_MB_BLK_COIL,
		Address     := 21889,
		pBlock      := ADR(MDB_Alarmes),
		blockLen    := SIZEOF(MDB_Alarmes)
	);
	mbusSetBlock(
        devIdent    := mbusDevice.devIdent,
        BlockType   := PGS_MB_BLK_COIL,
        Address     := 17089, (*50001*)
        pBlock      := ADR(MDB_Status),
        blockLen    := SIZEOF(MDB_Status)
    );
     mbusSetBlock(
        devIdent    := mbusDevice.devIdent,
        BlockType   := PGS_MB_BLK_COIL,
        Address     := 26689, (*50513*)
        pBlock      := ADR(MDB_Comandos),
        blockLen    := SIZEOF(MDB_Comandos)
    );

	    //Version
    mbusSetBlock(
        devIdent    := mbusDevice.devIdent,
        BlockType   := PGS_MB_BLK_INPUT,
        Address     := 65533,
        pBlock      := ADR(version),
        blockLen    := SIZEOF(version)
    );

    //TCP
    mbusTcpOpen (
        enable      := TRUE,
        dtaIdent    := mbusData.dtaIdent,
        port        := 502
    );
    mbusTcpUpdate.enable    := TRUE;
    mbusTcpUpdate.timeout   := 5.0;

    //Telnet
    telnetOpen (
        enable      := TRUE,
        port        := 23
    );
    telnetUpdate.enable    := TRUE;
    telnetUpdate.timeout   := 3600.0;

END_PROGRAM
```

### Program Logical/Auto/Auto

#### Init.st
```iecst
PROGRAM _INIT
	(* Insert code here *)
    TagManager(enable:=TRUE);
	//Registro de Parametros
    PgsTagStartNode     (TagManager.ident, ADR('Auto'));

    PgsTagStartNode     (TagManager.ident, ADR('Parametro'));
    PgsTagRegisterREAL  (TagManager.ident, TRUE, ADR('Var_par'),	Var_par);
    PgsTagEndNode       (TagManager.ident);//Parametro

	PgsTagStartNode     (TagManager.ident, ADR('Status'));
    PgsTagRegisterBOOL  (TagManager.ident, TRUE, ADR('Var_cmd'),	Var_cmd);
    PgsTagRegisterBOOL  (TagManager.ident, TRUE, ADR('dummy'),		dummy);
    PgsTagRegisterBOOL  (TagManager.ident, TRUE, ADR('dummy'),		dummy);
    PgsTagEndNode       (TagManager.ident);//Status

	PgsTagEndNode       (TagManager.ident);//Auto

END_PROGRAM
```

### Program Logical/Auto/Modbus/MDB_Comando (IEC)

#### Cyclic.st
```iecst
PROGRAM _CYCLIC
//********************************//
//** Coil register              **//
//** Função 01                  **//
//** Endereço 23000             **//
//** Tipo BOOL                  **//
//********************************//

//-------------------------------------------------------------------------------------------
//-- Trocar a variável "Var_cmd" por uma variável da automação ------------------------------
//-- Repetir a linha para todos os comandos, incrementando o número "01" a cada linha -------
//-------------------------------------------------------------------------------------------

	ExecutaComando(MDB_Comandos[01], Var_cmd);

//-------------------------------------------------------------------------------------------

END_PROGRAM
```

- Program Logical/Auto/Modbus/MDB_Alarme (IEC) (no source held here)

### Program Logical/Auto/Modbus/MDB_AL

#### Cyclic.st
```iecst
PROGRAM _CYCLIC

	//-------------------------------------------------------------------------------------------
	(*Alarmes*)
	//-------------------------------------------------------------------------------------------

	MDB_Alarmes[1] := UG.Alarme.UP_Partindo_Timeout;
	MDB_Alarmes[2] := UG.Alarme.UPGM_Partindo_Timeout;
	MDB_Alarmes[3] := UG.Alarme.UMVD_Partindo_Timeout;
	MDB_Alarmes[4] := UG.Alarme.UPS_Partindo_Timeout;
	MDB_Alarmes[5] := UG.Alarme.US_Parando_Timeout;
	MDB_Alarmes[6] := UG.Alarme.UPS_Parando_Timeout;
	MDB_Alarmes[7] := UG.Alarme.UMVD_Parando_Timeout;
	MDB_Alarmes[8] := UG.Alarme.UPGM_Parando_Timeout;
	MDB_Alarmes[9] := FALSE;
	MDB_Alarmes[10] := FALSE;
	MDB_Alarmes[11] := Painel.Alarme.CLP.Alim_IO;
	MDB_Alarmes[12] := Painel.Alarme.CLP.Alim_Modulo_01;
	MDB_Alarmes[13] := Painel.Alarme.CLP.Modulo_01;
	MDB_Alarmes[14] := Painel.Alarme.CLP.Modulo_02;
	MDB_Alarmes[15] := Painel.Alarme.CLP.Modulo_03;
	MDB_Alarmes[16] := Painel.Alarme.CLP.Modulo_04;
	MDB_Alarmes[17] := Painel.Alarme.CLP.Modulo_05;
	MDB_Alarmes[18] := Painel.Alarme.CLP.Modulo_06;
	MDB_Alarmes[19] := Painel.Alarme.CLP.Modulo_07;
	MDB_Alarmes[20] := Painel.Alarme.CLP.Modulo_08;
	MDB_Alarmes[21] := Painel.Alarme.CLP.Modulo_09;
	MDB_Alarmes[22] := Painel.Alarme.CLP.Modulo_10;
	MDB_Alarmes[23] := Painel.Alarme.CLP.Modulo_11;
	MDB_Alarmes[24] := Painel.Alarme.CLP.Modulo_12;
	MDB_Alarmes[25] := Painel.Alarme.CLP.Modulo_R1;
	MDB_Alarmes[26] := Painel.Alarme.CLP.Modulo_R2;
	MDB_Alarmes[27] := Painel.Alarme.CLP.Modulo_R3;
	MDB_Alarmes[28] := Painel.Alarme.CLP.Modulo_R4;
	MDB_Alarmes[29] := Painel.Alarme.CLP.Modulo_R5;
//	MDB_Alarmes[30] := Painel.Alarme.CLP.Modulo_18;
	MDB_Alarmes[31] := Painel.Alarme.CLP_Watchdog;
	MDB_Alarmes[32] := Painel.Alarme.RP_Watchdog;
	MDB_Alarmes[33] := Painel.Alarme.RP_Trip86E;
	MDB_Alarmes[34] := Painel.Alarme.RP_Trip86H;
	MDB_Alarmes[35] := Painel.Alarme.Emergencia;
	MDB_Alarmes[36] := Painel.Alarme.Emergencia_Remota;
	MDB_Alarmes[37] := Painel.Alarme.PSCP_Falta_tensao_VCC_Serv_Aux;
	MDB_Alarmes[38] := Painel.Alarme.QDAS_Falta_Tensao_125VCC;
	MDB_Alarmes[39] := Painel.Alarme.QDAS_DJ52_01_Aberto;
	MDB_Alarmes[40] := Painel.Alarme.Trafo_Exc_Fusivel_Queimado;
	MDB_Alarmes[41] := Painel.Alarme.Trafo_Exc_Temp_Alarme;
	MDB_Alarmes[42] := Painel.Alarme.Trafo_Exc_Temp_Trip;
	MDB_Alarmes[43] := Painel.Alarme.Trafo_Exc_Falha_Sensor;
	MDB_Alarmes[44] := Painel.Alarme.Falha.VCC_Ctrl_Prot;
	MDB_Alarmes[45] := Painel.Alarme.Trip_86E;
	MDB_Alarmes[46] := Painel.Alarme.Trip_86H;
	MDB_Alarmes[47] := Painel.Alarme.Trip_86M;
	MDB_Alarmes[48] := FALSE;
	MDB_Alarmes[49] := FALSE;
	MDB_Alarmes[50] := FALSE;
	MDB_Alarmes[51] := SFA.Alarme.Bomba1.Ligar;
	MDB_Alarmes[52] := SFA.Alarme.Bomba1.Desligar;
	MDB_Alarmes[53] := SFA.Alarme.DJM.Trip;
	MDB_Alarmes[54] := SFA.Alarme.Filtro1_Lado_Limpo.Cabo_Aberto;
	MDB_Alarmes[55] := SFA.Alarme.Filtro1_Lado_Limpo.Cabo_Curto;
	MDB_Alarmes[56] := SFA.Alarme.Filtro1_Lado_Sujo.Cabo_Aberto;
	MDB_Alarmes[57] := SFA.Alarme.Filtro1_Lado_Sujo.Cabo_Curto;
	MDB_Alarmes[58] := SFA.Alarme.Filtro1_Sujo; //Alarme diferencial de pressão filtro1 - 500 micra
	MDB_Alarmes[59] := SFA.Alarme.Pressao.Trip;
	MDB_Alarmes[60] := SFA.Alarme.Filtro2_Lado_Limpo.Cabo_Aberto;
	MDB_Alarmes[61] := SFA.Alarme.Filtro2_Lado_Limpo.Cabo_Curto;
	MDB_Alarmes[62] := SFA.Alarme.Filtro2_Lado_Sujo.Cabo_Aberto;
	MDB_Alarmes[63] := SFA.Alarme.Filtro2_Lado_Sujo.Cabo_Curto;
	MDB_Alarmes[64] := SFA.Alarme.Filtro2_Sujo; //Alarme diferencial de pressão filtro2 - 50 micra
	MDB_Alarmes[65] := FALSE;
	MDB_Alarmes[66] := FALSE;
	MDB_Alarmes[67] := FALSE;
	MDB_Alarmes[68] := FALSE;
	MDB_Alarmes[69] := FALSE;
	MDB_Alarmes[70] := FALSE;
	MDB_Alarmes[71] := UHLM.Alarme.Bomba1.Ligar;
	MDB_Alarmes[72] := UHLM.Alarme.Bomba1.Desligar;
	MDB_Alarmes[73] := UHLM.Alarme.Bomba1.DJM.Trip;
	MDB_Alarmes[74] := UHLM.Alarme.Bomba2.Ligar;
	MDB_Alarmes[75] := UHLM.Alarme.Bomba2.Desligar;
	MDB_Alarmes[76] := UHLM.Alarme.Bomba2.DJM.Trip;
	MDB_Alarmes[77] := UHLM.Alarme.JackingOil.Ligar;
	MDB_Alarmes[78] := UHLM.Alarme.JackingOil.Desligar;
	MDB_Alarmes[79] := UHLM.Alarme.JackingOil.DJM.Trip;
	MDB_Alarmes[80] := UHLM.Alarme.Ventilador.Ligar;
	MDB_Alarmes[81] := UHLM.Alarme.Ventilador.Desligar;
	MDB_Alarmes[82] := UHLM.Alarme.Ventilador.DJM.Trip;
	MDB_Alarmes[83] := UHLM.Alarme.Nivel_Minimo;
	MDB_Alarmes[84] := UHLM.Alarme.Nivel_Maximo;
	MDB_Alarmes[85] := UHLM.Alarme.Temperatura.Alarme;
	MDB_Alarmes[86] := UHLM.Alarme.Temperatura.Trip;
	MDB_Alarmes[87] := UHLM.Alarme.Temperatura.Cabo_Aberto;
	MDB_Alarmes[88] := UHLM.Alarme.Temperatura.Cabo_Curto;
	MDB_Alarmes[89] := UHLM.Alarme.Vazao.Alarme;
	MDB_Alarmes[90] := UHLM.Alarme.Vazao.Trip;
	MDB_Alarmes[91] := UHLM.Alarme.Vazao.Cabo_Aberto;
	MDB_Alarmes[92] := UHLM.Alarme.Vazao.Cabo_Curto;
	MDB_Alarmes[93] := UHLM.Alarme.Fluxo1.Trip;(*Fluxostato trocador de calor mancal combinado*)
	MDB_Alarmes[94] := UHLM.Alarme.Fluxo2.Trip;(*Fluxostato trocador de calor mancal guia*)
//	MDB_Alarmes[95] := UHLM.Alarme.Fluxo3.Trip;
//	MDB_Alarmes[96] := UHLM.Alarme.Fluxo4.Trip;
//	MDB_Alarmes[97] := UHLM.Alarme.Fluxo5.Trip;
	MDB_Alarmes[98] := UHLM.Alarme.Pressao1.Trip;(*Pressostato linha jacking oil*)
	MDB_Alarmes[99] := UHLM.Alarme.Pressao2.Trip;(*Pressostato mancal combinado*)
	MDB_Alarmes[100] := UHLM.Alarme.Pressao3.Trip;(*Pressostato mancal guia*)
//	MDB_Alarmes[101] := UHLM.Alarme.Pressao4.Trip;
//	MDB_Alarmes[102] := UHLM.Alarme.Pressao5.Trip;
	MDB_Alarmes[103] := UHLM.Alarme.Filtro_Sujo1;(*Filtro sujo linha do jacking oil*)
	MDB_Alarmes[104] := UHLM.Alarme.Filtro_Sujo2;(*Filtro sujo linha do mancal combinado*)
	MDB_Alarmes[105] := UHLM.Alarme.Filtro_Sujo3;(*Filtro sujo linha do mancal guia*)
	MDB_Alarmes[106] := UHLM.Alarme.Mancal_Guia_Nivel_Min;
	MDB_Alarmes[107] := UHLM.Alarme.Mancal_Guia_Nivel_Max;
	MDB_Alarmes[108] := UHLM.Alarme.Bomba3.Ligar;
	MDB_Alarmes[109] := UHLM.Alarme.Bomba3.Desligar;
	MDB_Alarmes[110] := UHLM.Alarme.Bomba3.DJM.Trip;
	MDB_Alarmes[111] := UHRV.Alarme.Bomba1.Ligar;
	MDB_Alarmes[112] := UHRV.Alarme.Bomba1.Desligar;
	MDB_Alarmes[113] := UHRV.Alarme.Bomba1.DJM.Trip;
	MDB_Alarmes[114] := UHRV.Alarme.Bomba2.Ligar;
	MDB_Alarmes[115] := UHRV.Alarme.Bomba2.Desligar;
	MDB_Alarmes[116] := UHRV.Alarme.Bomba2.DJM.Trip;
//	MDB_Alarmes[117] := UHRV.Alarme.Bomba3.Ligar;
//	MDB_Alarmes[118] := UHRV.Alarme.Bomba3.Desligar;
//	MDB_Alarmes[119] := UHRV.Alarme.Bomba3.DJM.Trip;
//	MDB_Alarmes[120] := UHRV.Alarme.Ventilador.Ligar;
//	MDB_Alarmes[121] := UHRV.Alarme.Ventilador.Desligar;
//	MDB_Alarmes[122] := UHRV.Alarme.Ventilador.DJM.Trip;
	MDB_Alarmes[123] := UHRV.Alarme.Filtro1.Pressao.Sujo;
	MDB_Alarmes[124] := UHRV.Alarme.Filtro1.Pressao.Saturado;
	MDB_Alarmes[125] := UHRV.Alarme.Filtro2.Pressao.Sujo;
	MDB_Alarmes[126] := UHRV.Alarme.Filtro2.Pressao.Saturado;
	MDB_Alarmes[127] := UHRV.Alarme.Filtro1.Retorno.Sujo;
	MDB_Alarmes[128] := UHRV.Alarme.Filtro1.Retorno.Saturado;
	MDB_Alarmes[129] := UHRV.Alarme.Filtro2.Retorno.Sujo;
	MDB_Alarmes[130] := UHRV.Alarme.Filtro2.Retorno.Saturado;
	MDB_Alarmes[131] := UHRV.Alarme.Nivel.Maximo;
	MDB_Alarmes[132] := UHRV.Alarme.Nivel.Minimo;
	MDB_Alarmes[133] := UHRV.Alarme.Nivel.Critico;
	MDB_Alarmes[134] := UHRV.Alarme.Temperatura.Alarme;
	MDB_Alarmes[135] := UHRV.Alarme.Temperatura.Trip;
	MDB_Alarmes[136] := UHRV.Alarme.Temperatura.Cabo_Aberto;
	MDB_Alarmes[137] := UHRV.Alarme.Temperatura.Cabo_Curto;
	MDB_Alarmes[138] := UHRV.Alarme.Pressao.Alarme;
	MDB_Alarmes[139] := UHRV.Alarme.Pressao.Trip;
	MDB_Alarmes[140] := UHRV.Alarme.Pressao.Cabo_Aberto;
	MDB_Alarmes[141] := UHRV.Alarme.Pressao.Cabo_Curto;
	MDB_Alarmes[142] := UHRV.Alarme.Pressostato.Maxima;
	MDB_Alarmes[143] := UHRV.Alarme.Pressostato.Minima;
	MDB_Alarmes[144] := UHRV.Alarme.Pressao_Critica;
	MDB_Alarmes[145] := UHRV.Alarme.Pressurizar;
	MDB_Alarmes[146] := FALSE;
	MDB_Alarmes[147] := FALSE;
	MDB_Alarmes[148] := FALSE;
	MDB_Alarmes[149] := FALSE;
	MDB_Alarmes[150] := FALSE;
	MDB_Alarmes[151] := FALSE;
	MDB_Alarmes[152] := FALSE;
	MDB_Alarmes[153] := FALSE;
	MDB_Alarmes[154] := FALSE;
	MDB_Alarmes[155] := FALSE;
	MDB_Alarmes[156] := FALSE;
	MDB_Alarmes[157] := FALSE;
	MDB_Alarmes[158] := FALSE;
	MDB_Alarmes[159] := FALSE;
	MDB_Alarmes[160] := FALSE;
	MDB_Alarmes[161] := Freio.Alarme.Aplicar;
	MDB_Alarmes[162] := Freio.Alarme.Desaplicar;
	MDB_Alarmes[163] := Freio.Alarme.Pressostato_Critica;
	MDB_Alarmes[164] := Freio.Alarme.Pastilhas_Gastas;
	MDB_Alarmes[165] := Freio.Alarme.Inconsistente;
//	MDB_Alarmes[166] := Freio.Alarme.Falta_Pressao;(*ok*)
	MDB_Alarmes[167] := FALSE;
	MDB_Alarmes[168] := FALSE;
	MDB_Alarmes[169] := FALSE;
	MDB_Alarmes[170] := FALSE;
//	MDB_Alarmes[171] := VByPass.Alarme.Abrir;
//	MDB_Alarmes[172] := VByPass.Alarme.Fechar;
	MDB_Alarmes[173] := FALSE;
	MDB_Alarmes[174] := FALSE;
	MDB_Alarmes[175] := FALSE;
	MDB_Alarmes[176] := FALSE;
	MDB_Alarmes[177] := FALSE;
	MDB_Alarmes[178] := FALSE;
	MDB_Alarmes[179] := FALSE;
	MDB_Alarmes[180] := FALSE;
//	MDB_Alarmes[181] := VBorb.Alarme.Abrir;
//	MDB_Alarmes[182] := VBorb.Alarme.Fechar;
//	MDB_Alarmes[183] := VBorb.Alarme.Equalizar;
//	MDB_Alarmes[184] := VBorb.Alarme.Reposicao;
	MDB_Alarmes[185] := Comporta_UH.Alarme.Nivel_Critico;
	MDB_Alarmes[186] := Comporta_UH.Alarme.Pressao_Ruptura;
	MDB_Alarmes[187] := Comporta1.Alarme.Encoder1_Cabo_Aberto;
	MDB_Alarmes[188] := Comporta1.Alarme.Encoder1_Cabo_Curto;
	MDB_Alarmes[189] := Comporta2.Alarme.Encoder2_Cabo_Aberto;
	MDB_Alarmes[190] := Comporta2.Alarme.Encoder2_Cabo_Curto;
	MDB_Alarmes[191] := Comportas.Alarme_Bloqueio_Comando_Local;
	MDB_Alarmes[192] := Comporta_UH.Alarme.Filtro.Sujo;
	MDB_Alarmes[193] := Comporta_UH.Alarme.Comandos_Desligados;
	MDB_Alarmes[194] := Comporta_UH.Alarme.Falha_Tensao_380V;
	MDB_Alarmes[195] := Comporta1.Alarme.Deriva;
	MDB_Alarmes[196] := Comporta2.Alarme.Deriva;
	MDB_Alarmes[197] := Comporta_UH.Alarme.Bomba1.DJM.Trip;
	MDB_Alarmes[198] := Comporta_UH.Alarme.Bomba2.DJM.Trip;
	MDB_Alarmes[199] := Comporta_UH.Alarme.Pressao_Alta;
	MDB_Alarmes[200] := Comporta_UH.Alarme.Pressao_Baixa;
	MDB_Alarmes[201] := Comporta1.Alarme.Timeout_Abertura;
	MDB_Alarmes[202] := Comporta1.Alarme.Timeout_Fechando;
	MDB_Alarmes[203] := Comporta1.Alarme.Timeout_Cracking;
	MDB_Alarmes[204] := Comporta1.Alarme.Timeout_Reposicao;
	MDB_Alarmes[205] := Comporta1.Alarme.Falha_Cracking;
	MDB_Alarmes[206] := Comporta1.Alarme.Falha_Reposicao;
	MDB_Alarmes[207] := Comporta_UH.Alarme.Temperatura.Cabo_Aberto;
	MDB_Alarmes[208] := Comporta_UH.Alarme.Temperatura.Cabo_Curto;
	MDB_Alarmes[209] := Comporta_UH.Alarme.Temperatura.Alarme;
	MDB_Alarmes[210] := Comporta_UH.Alarme.Temperatura.Trip;
	MDB_Alarmes[211] := Comporta2.Alarme.Timeout_Abertura;
	MDB_Alarmes[212] := Comporta2.Alarme.Timeout_Fechando;
	MDB_Alarmes[213] := Comporta2.Alarme.Timeout_Cracking;
	MDB_Alarmes[214] := Comporta2.Alarme.Timeout_Reposicao;
	MDB_Alarmes[215] := Comporta2.Alarme.Falha_Cracking;
	MDB_Alarmes[216] := Comporta2.Alarme.Falha_Reposicao;
	MDB_Alarmes[217] := Comporta_UH.Alarme.Bomba1.Ligar;
	MDB_Alarmes[218] := Comporta_UH.Alarme.Bomba2.Ligar;
	MDB_Alarmes[219] := Comporta_UH.Alarme.Nivel_Baixo;
	MDB_Alarmes[220] := Comporta_UH.Alarme.Nivel_Alto;
	MDB_Alarmes[221] := Turbina.Alarme.Sobre_Velocidade_Mecanico;
	MDB_Alarmes[222] := Turbina.Alarme.Gaxeteiro.Temperatura.Alarme;
	MDB_Alarmes[223] := Turbina.Alarme.Gaxeteiro.Temperatura.Trip;
	MDB_Alarmes[224] := Turbina.Alarme.Gaxeteiro.Temperatura.Cabo_Aberto;
	MDB_Alarmes[225] := Turbina.Alarme.Gaxeteiro.Temperatura.Cabo_Curto;
	MDB_Alarmes[226] := Turbina.Alarme.Mancal1.Temperatura.Alarme;
	MDB_Alarmes[227] := Turbina.Alarme.Mancal1.Temperatura.Trip;
	MDB_Alarmes[228] := Turbina.Alarme.Mancal1.Temperatura.Cabo_Aberto;
	MDB_Alarmes[229] := Turbina.Alarme.Mancal1.Temperatura.Cabo_Curto;
	MDB_Alarmes[230] := Turbina.Alarme.Mancal2.Temperatura.Alarme;
	MDB_Alarmes[231] := Turbina.Alarme.Mancal2.Temperatura.Trip;
	MDB_Alarmes[232] := Turbina.Alarme.Mancal2.Temperatura.Cabo_Aberto;
	MDB_Alarmes[233] := Turbina.Alarme.Mancal2.Temperatura.Cabo_Curto;
	MDB_Alarmes[234] := Turbina.Alarme.Mancal3.Temperatura.Alarme;
	MDB_Alarmes[235] := Turbina.Alarme.Mancal3.Temperatura.Trip;
	MDB_Alarmes[236] := Turbina.Alarme.Mancal3.Temperatura.Cabo_Aberto;
	MDB_Alarmes[237] := Turbina.Alarme.Mancal3.Temperatura.Cabo_Curto;
	MDB_Alarmes[238] := Turbina.Alarme.Mancal4.Temperatura.Alarme;
	MDB_Alarmes[239] := Turbina.Alarme.Mancal4.Temperatura.Trip;
	MDB_Alarmes[240] := Turbina.Alarme.Mancal4.Temperatura.Cabo_Aberto;
	MDB_Alarmes[241] := Turbina.Alarme.Mancal4.Temperatura.Cabo_Curto;
	MDB_Alarmes[242] := Turbina.Alarme.Mancal5.Temperatura.Alarme;
	MDB_Alarmes[243] := Turbina.Alarme.Mancal5.Temperatura.Trip;
	MDB_Alarmes[244] := Turbina.Alarme.Mancal5.Temperatura.Cabo_Aberto;
	MDB_Alarmes[245] := Turbina.Alarme.Mancal5.Temperatura.Cabo_Curto;
	MDB_Alarmes[246] := Turbina.Alarme.Mancal6.Temperatura.Alarme;
	MDB_Alarmes[247] := Turbina.Alarme.Mancal6.Temperatura.Trip;
	MDB_Alarmes[248] := Turbina.Alarme.Mancal6.Temperatura.Cabo_Aberto;
	MDB_Alarmes[249] := Turbina.Alarme.Mancal6.Temperatura.Cabo_Curto;
	MDB_Alarmes[250] := Turbina.Alarme.CaixaEspiral.Pressao.Alarme;
	MDB_Alarmes[251] := Turbina.Alarme.CaixaEspiral.Pressao.Trip;
	MDB_Alarmes[252] := Turbina.Alarme.CaixaEspiral.Pressao.Cabo_Aberto;
	MDB_Alarmes[253] := Turbina.Alarme.CaixaEspiral.Pressao.Cabo_Curto;
	MDB_Alarmes[254] := Turbina.Alarme.Boia_Selo_Agua_TRIP;
	MDB_Alarmes[255] := Turbina.Alarme.Pas_Desalinha;
	MDB_Alarmes[256] := FALSE;
	MDB_Alarmes[257] := FALSE;
	MDB_Alarmes[258] := FALSE;
	MDB_Alarmes[259] := FALSE;
	MDB_Alarmes[260] := FALSE;
	MDB_Alarmes[261] := FALSE;
	MDB_Alarmes[262] := FALSE;
	MDB_Alarmes[263] := FALSE;
	MDB_Alarmes[264] := FALSE;
	MDB_Alarmes[265] := FALSE;
	MDB_Alarmes[266] := FALSE;
	MDB_Alarmes[267] := FALSE;
	MDB_Alarmes[268] := FALSE;
	MDB_Alarmes[269] := FALSE;
	MDB_Alarmes[270] := FALSE;
	MDB_Alarmes[271] := Gerador.Alarme.Fase_A.Temperatura.Alarme;
	MDB_Alarmes[272] := Gerador.Alarme.Fase_A.Temperatura.Trip;
	MDB_Alarmes[273] := Gerador.Alarme.Fase_A.Temperatura.Cabo_Aberto;
	MDB_Alarmes[274] := Gerador.Alarme.Fase_A.Temperatura.Cabo_Curto;
	MDB_Alarmes[275] := Gerador.Alarme.Fase_B.Temperatura.Alarme;
	MDB_Alarmes[276] := Gerador.Alarme.Fase_B.Temperatura.Trip;
	MDB_Alarmes[277] := Gerador.Alarme.Fase_B.Temperatura.Cabo_Aberto;
	MDB_Alarmes[278] := Gerador.Alarme.Fase_B.Temperatura.Cabo_Curto;
	MDB_Alarmes[279] := Gerador.Alarme.Fase_C.Temperatura.Alarme;
	MDB_Alarmes[280] := Gerador.Alarme.Fase_C.Temperatura.Trip;
	MDB_Alarmes[281] := Gerador.Alarme.Fase_C.Temperatura.Cabo_Aberto;
	MDB_Alarmes[282] := Gerador.Alarme.Fase_C.Temperatura.Cabo_Curto;
	MDB_Alarmes[283] := Gerador.Alarme.NucleoEstatorico1.Temperatura.Alarme;
	MDB_Alarmes[284] := Gerador.Alarme.NucleoEstatorico1.Temperatura.Trip;
	MDB_Alarmes[285] := Gerador.Alarme.NucleoEstatorico1.Temperatura.Cabo_Aberto;
	MDB_Alarmes[286] := Gerador.Alarme.NucleoEstatorico1.Temperatura.Cabo_Curto;
	MDB_Alarmes[287] := Gerador.Alarme.NucleoEstatorico2.Temperatura.Alarme;
	MDB_Alarmes[288] := Gerador.Alarme.NucleoEstatorico2.Temperatura.Trip;
	MDB_Alarmes[289] := Gerador.Alarme.NucleoEstatorico2.Temperatura.Cabo_Aberto;
	MDB_Alarmes[290] := Gerador.Alarme.NucleoEstatorico2.Temperatura.Cabo_Curto;
	MDB_Alarmes[291] := Gerador.Alarme.NucleoEstatorico3.Temperatura.Alarme;
	MDB_Alarmes[292] := Gerador.Alarme.NucleoEstatorico3.Temperatura.Trip;
	MDB_Alarmes[293] := Gerador.Alarme.NucleoEstatorico3.Temperatura.Cabo_Aberto;
	MDB_Alarmes[294] := Gerador.Alarme.NucleoEstatorico3.Temperatura.Cabo_Curto;
	MDB_Alarmes[295] := Gerador.Alarme.Mancal1.Temperatura.Alarme;
	MDB_Alarmes[296] := Gerador.Alarme.Mancal1.Temperatura.Trip;
	MDB_Alarmes[297] := Gerador.Alarme.Mancal1.Temperatura.Cabo_Aberto;
	MDB_Alarmes[298] := Gerador.Alarme.Mancal1.Temperatura.Cabo_Curto;
	MDB_Alarmes[299] := Gerador.Alarme.Mancal2.Temperatura.Alarme;
	MDB_Alarmes[300] := Gerador.Alarme.Mancal2.Temperatura.Trip;
	MDB_Alarmes[301] := Gerador.Alarme.Mancal2.Temperatura.Cabo_Aberto;
	MDB_Alarmes[302] := Gerador.Alarme.Mancal2.Temperatura.Cabo_Curto;
	MDB_Alarmes[303] := Gerador.Alarme.Mancal3.Temperatura.Alarme;
	MDB_Alarmes[304] := Gerador.Alarme.Mancal3.Temperatura.Trip;
	MDB_Alarmes[305] := Gerador.Alarme.Mancal3.Temperatura.Cabo_Aberto;
	MDB_Alarmes[306] := Gerador.Alarme.Mancal3.Temperatura.Cabo_Curto;
	MDB_Alarmes[307] := Gerador.Alarme.Mancal4.Temperatura.Alarme;
	MDB_Alarmes[308] := Gerador.Alarme.Mancal4.Temperatura.Trip;
	MDB_Alarmes[309] := Gerador.Alarme.Mancal4.Temperatura.Cabo_Aberto;
	MDB_Alarmes[310] := Gerador.Alarme.Mancal4.Temperatura.Cabo_Curto;
	MDB_Alarmes[311] := Gerador.Alarme.Mancal5.Temperatura.Alarme;
	MDB_Alarmes[312] := Gerador.Alarme.Mancal5.Temperatura.Trip;
	MDB_Alarmes[313] := Gerador.Alarme.Mancal5.Temperatura.Cabo_Aberto;
	MDB_Alarmes[314] := Gerador.Alarme.Mancal5.Temperatura.Cabo_Curto;
	MDB_Alarmes[315] := Gerador.Alarme.Mancal6.Temperatura.Alarme;
	MDB_Alarmes[316] := Gerador.Alarme.Mancal6.Temperatura.Trip;
	MDB_Alarmes[317] := Gerador.Alarme.Mancal6.Temperatura.Cabo_Aberto;
	MDB_Alarmes[318] := Gerador.Alarme.Mancal6.Temperatura.Cabo_Curto;
	MDB_Alarmes[319] := Gerador.Alarme.Escovas_Gastas_Neg;(*OK*)
	MDB_Alarmes[320] := Gerador.Alarme.Escovas_Gastas_Pos;(*OK*)
	MDB_Alarmes[321] := FALSE;
	MDB_Alarmes[322] := FALSE;
	MDB_Alarmes[323] := FALSE;
	MDB_Alarmes[324] := FALSE;
	MDB_Alarmes[325] := FALSE;
	MDB_Alarmes[326] := FALSE;
	MDB_Alarmes[327] := FALSE;
	MDB_Alarmes[328] := FALSE;
	MDB_Alarmes[329] := FALSE;
	MDB_Alarmes[330] := FALSE;
	MDB_Alarmes[331] := FALSE;
	MDB_Alarmes[332] := FALSE;
	MDB_Alarmes[333] := FALSE;
	MDB_Alarmes[334] := FALSE;
	MDB_Alarmes[335] := FALSE;
	MDB_Alarmes[336] := FALSE;
	MDB_Alarmes[337] := FALSE;
	MDB_Alarmes[338] := FALSE;
	MDB_Alarmes[339] := FALSE;
	MDB_Alarmes[340] := FALSE;
	MDB_Alarmes[341] := RT.Alarme.Crowbar;
	MDB_Alarmes[342] := RT.Alarme.DJ_Field_Flash.Trip;
	MDB_Alarmes[343] := RT.Alarme.PWR.Termostato.Alarme;
	MDB_Alarmes[344] := RT.Alarme.PWR.Termostato.Trip;
	MDB_Alarmes[345] := RT.Alarme.PWR.Temperatura.Alarme;
	MDB_Alarmes[346] := RT.Alarme.PWR.Temperatura.Trip;
	MDB_Alarmes[347] := RT.Alarme.PWR.Temperatura.Cabo_Aberto;
	MDB_Alarmes[348] := RT.Alarme.PWR.Temperatura.Cabo_Curto;
	MDB_Alarmes[349] := RT.Alarme.PWR.Fusivel_Queimado;
	MDB_Alarmes[350] := FALSE;
	MDB_Alarmes[351] := FALSE;
	MDB_Alarmes[352] := FALSE;
	MDB_Alarmes[353] := FALSE;
	MDB_Alarmes[354] := FALSE;
	MDB_Alarmes[355] := FALSE;
	MDB_Alarmes[356] := FALSE;
	MDB_Alarmes[357] := FALSE;
	MDB_Alarmes[358] := FALSE;
	MDB_Alarmes[359] := FALSE;
	MDB_Alarmes[360] := FALSE;
	MDB_Alarmes[361] := Trafo_Exc.Alarme.Fase_A.Temperatura.Alarme;
	MDB_Alarmes[362] := Trafo_Exc.Alarme.Fase_A.Temperatura.Trip;
	MDB_Alarmes[363] := Trafo_Exc.Alarme.Fase_A.Temperatura.Cabo_Aberto;
	MDB_Alarmes[364] := Trafo_Exc.Alarme.Fase_A.Temperatura.Cabo_Curto;
	MDB_Alarmes[365] := Trafo_Exc.Alarme.Fase_B.Temperatura.Alarme;
	MDB_Alarmes[366] := Trafo_Exc.Alarme.Fase_B.Temperatura.Trip;
	MDB_Alarmes[367] := Trafo_Exc.Alarme.Fase_B.Temperatura.Cabo_Aberto;
	MDB_Alarmes[368] := Trafo_Exc.Alarme.Fase_B.Temperatura.Cabo_Curto;
	MDB_Alarmes[369] := Trafo_Exc.Alarme.Fase_C.Temperatura.Alarme;
	MDB_Alarmes[370] := Trafo_Exc.Alarme.Fase_C.Temperatura.Trip;
	MDB_Alarmes[371] := Trafo_Exc.Alarme.Fase_C.Temperatura.Cabo_Aberto;
	MDB_Alarmes[372] := Trafo_Exc.Alarme.Fase_C.Temperatura.Cabo_Curto;
	MDB_Alarmes[373] := Trafo_Exc.Alarme.Fusiveis_Queimados;
	MDB_Alarmes[374] := Trafo_Exc.Alarme.Falha_Sensor_Temp;
	MDB_Alarmes[375] := Trafo_Exc.Alarme.Temperatura_Alarme;
	MDB_Alarmes[376] := Trafo_Exc.Alarme.Temperatura_Trip;
	MDB_Alarmes[377] := FALSE;
	MDB_Alarmes[378] := FALSE;
	MDB_Alarmes[379] := FALSE;
	MDB_Alarmes[380] := FALSE;
	MDB_Alarmes[381] := DJ52G.Alarme.Inconsistente;
//	MDB_Alarmes[382] := DJ52L.Alarme.Inconsistente;
	MDB_Alarmes[383] := DJ52G.Alarme.Falha;
	MDB_Alarmes[384] := DJ52G.Alarme.Extraido;
	MDB_Alarmes[385] := DJ52G.Alarme.Modo_Teste;
	MDB_Alarmes[386] := DJ52G.Alarme.Falta_125Vcc;
	MDB_Alarmes[387] := FALSE;
	MDB_Alarmes[388] := FALSE;
	MDB_Alarmes[389] := FALSE;
	MDB_Alarmes[390] := FALSE;
	MDB_Alarmes[391] := Nivel.Alarme.Nivel_Desligar;
	MDB_Alarmes[392] := Nivel.Alarme.Nivel_Trip;
	MDB_Alarmes[393] := Nivel.Alarme.Barragem.Cabo_Aberto;
	MDB_Alarmes[394] := Nivel.Alarme.Barragem.Cabo_Curto;
	MDB_Alarmes[395] := Nivel.Alarme.Jusante_Grade1.Alarme;
	MDB_Alarmes[396] := Nivel.Alarme.Jusante_Grade1.Trip;
	MDB_Alarmes[397] := Nivel.Alarme.Jusante_Grade1.Cabo_Aberto;
	MDB_Alarmes[398] := Nivel.Alarme.Jusante_Grade1.Cabo_Curto;
	MDB_Alarmes[399] := Nivel.Alarme.Jusante_Grade2.Alarme;
	MDB_Alarmes[400] := Nivel.Alarme.Jusante_Grade2.Trip;
	MDB_Alarmes[401] := Nivel.Alarme.Jusante_Grade2.Cabo_Aberto;
	MDB_Alarmes[402] := Nivel.Alarme.Jusante_Grade2.Cabo_Curto;
	MDB_Alarmes[403] := Nivel.Alarme.Jusante.Alarme;
	MDB_Alarmes[404] := Nivel.Alarme.Jusante.Trip;
	MDB_Alarmes[405] := Nivel.Alarme.Jusante.Cabo_Aberto;
	MDB_Alarmes[406] := Nivel.Alarme.Jusante.Cabo_Curto;
	MDB_Alarmes[407] := FALSE;
	MDB_Alarmes[408] := FALSE;
	MDB_Alarmes[409] := FALSE;
	MDB_Alarmes[410] := FALSE;
	MDB_Alarmes[411] := FALSE;
	MDB_Alarmes[412] := FALSE;
	MDB_Alarmes[413] := FALSE;
	MDB_Alarmes[414] := FALSE;
	MDB_Alarmes[415] := FALSE;
	MDB_Alarmes[416] := FALSE;
	MDB_Alarmes[417] := FALSE;
	MDB_Alarmes[418] := FALSE;
	MDB_Alarmes[419] := FALSE;
	MDB_Alarmes[420] := FALSE;
	MDB_Alarmes[421] := FALSE;
	MDB_Alarmes[422] := FALSE;
	MDB_Alarmes[423] := FALSE;
	MDB_Alarmes[424] := FALSE;

	//-------------------------------------------------------------------------------------------
END_PROGRAM
```

### Program Logical/Auto/Modbus/MDB_CMD (IEC)

#### Cyclic.st - Cyclic code
```iecst
PROGRAM _CYCLIC

	//-------------------------------------------------------------------------------------------
    (*Comandos*)
	//-------------------------------------------------------------------------------------------

	ExecutaComando(MDB_Comandos[1], UG.Comando.Local.Modo.Automatico);
	ExecutaComando(MDB_Comandos[2], UG.Comando.Local.Modo.Manual);
	ExecutaComando(MDB_Comandos[3], UG.Comando.Local.Modo.Manutencao);
	ExecutaComando(MDB_Comandos[4], UG.Comando.Local.Auto.UP);
	ExecutaComando(MDB_Comandos[5], UG.Comando.Local.Auto.UPGM);
	ExecutaComando(MDB_Comandos[6], UG.Comando.Local.Auto.UMVD);
	ExecutaComando(MDB_Comandos[7], UG.Comando.Local.Auto.UPS);
	ExecutaComando(MDB_Comandos[8], UG.Comando.Local.Auto.US);
	ExecutaComando(MDB_Comandos[9], UG.Comando.Local.Manual.SFA.Habilitar);
	ExecutaComando(MDB_Comandos[10], UG.Comando.Local.Manual.SFA.Desabilitar);
	ExecutaComando(MDB_Comandos[11], UG.Comando.Local.Manual.UHLM.Habilitar);
	ExecutaComando(MDB_Comandos[12], UG.Comando.Local.Manual.UHLM.Desabilitar);
	ExecutaComando(MDB_Comandos[13], UG.Comando.Local.Manual.UHRV.Habilitar);
	ExecutaComando(MDB_Comandos[14], UG.Comando.Local.Manual.UHRV.Desabilitar);
	ExecutaComando(MDB_Comandos[15], UG.Comando.Local.Manual.Freio.Habilitar);
	ExecutaComando(MDB_Comandos[16], UG.Comando.Local.Manual.Freio.Desabilitar);
//	ExecutaComando(MDB_Comandos[17], UG.Comando.Local.Manual.VByPass.Abrir);
//	ExecutaComando(MDB_Comandos[18], UG.Comando.Local.Manual.VByPass.Fechar);
//	ExecutaComando(MDB_Comandos[19], UG.Comando.Local.Manual.Vborb.Abrir);
//	ExecutaComando(MDB_Comandos[20], UG.Comando.Local.Manual.Vborb.Fechar);
	ExecutaComando(MDB_Comandos[21], UG.Comando.Local.Manual.Comporta1.Abrir);
	ExecutaComando(MDB_Comandos[22], UG.Comando.Local.Manual.Comporta1.Fechar);
	ExecutaComando(MDB_Comandos[23], UG.Comando.Local.Manual.Comporta2.Abrir);
	ExecutaComando(MDB_Comandos[24], UG.Comando.Local.Manual.Comporta2.Fechar);
	ExecutaComando(MDB_Comandos[25], UG.Comando.Local.Manual.RV.Habilitar);
	ExecutaComando(MDB_Comandos[26], UG.Comando.Local.Manual.RV.Desabilitar);
	ExecutaComando(MDB_Comandos[27], UG.Comando.Local.Manual.RT.Habilitar);
	ExecutaComando(MDB_Comandos[28], UG.Comando.Local.Manual.RT.Desabilitar);
	ExecutaComando(MDB_Comandos[29], UG.Comando.Local.Manual.SC.Habilitar);
	ExecutaComando(MDB_Comandos[30], UG.Comando.Local.Manual.SC.Desabilitar);
//	ExecutaComando(MDB_Comandos[31], FALSE);
//	ExecutaComando(MDB_Comandos[32], FALSE);
//	ExecutaComando(MDB_Comandos[33], FALSE);
//	ExecutaComando(MDB_Comandos[34], FALSE);
//	ExecutaComando(MDB_Comandos[35], FALSE);
//	ExecutaComando(MDB_Comandos[36], FALSE);
//	ExecutaComando(MDB_Comandos[37], FALSE);
//	ExecutaComando(MDB_Comandos[38], FALSE);
//	ExecutaComando(MDB_Comandos[39], FALSE);
//	ExecutaComando(MDB_Comandos[40], FALSE);
	ExecutaComando(MDB_Comandos[41], UG.Comando.Remoto.Modo.Automatico);
	ExecutaComando(MDB_Comandos[42], UG.Comando.Remoto.Modo.Manual);
	ExecutaComando(MDB_Comandos[43], UG.Comando.Remoto.Modo.Manutencao);
	ExecutaComando(MDB_Comandos[44], UG.Comando.Remoto.Auto.UP);
	ExecutaComando(MDB_Comandos[45], UG.Comando.Remoto.Auto.UPGM);
	ExecutaComando(MDB_Comandos[46], UG.Comando.Remoto.Auto.UMVD);
	ExecutaComando(MDB_Comandos[47], UG.Comando.Remoto.Auto.UPS);
	ExecutaComando(MDB_Comandos[48], UG.Comando.Remoto.Auto.US);
	ExecutaComando(MDB_Comandos[49], UG.Comando.Remoto.Manual.SFA.Habilitar);
	ExecutaComando(MDB_Comandos[50], UG.Comando.Remoto.Manual.SFA.Desabilitar);
	ExecutaComando(MDB_Comandos[51], UG.Comando.Remoto.Manual.UHLM.Habilitar);
	ExecutaComando(MDB_Comandos[52], UG.Comando.Remoto.Manual.UHLM.Desabilitar);
	ExecutaComando(MDB_Comandos[53], UG.Comando.Remoto.Manual.UHRV.Habilitar);
	ExecutaComando(MDB_Comandos[54], UG.Comando.Remoto.Manual.UHRV.Desabilitar);
	ExecutaComando(MDB_Comandos[55], UG.Comando.Remoto.Manual.Freio.Habilitar);
	ExecutaComando(MDB_Comandos[56], UG.Comando.Remoto.Manual.Freio.Desabilitar);
//	ExecutaComando(MDB_Comandos[57], UG.Comando.Remoto.Manual.VByPass.Abrir);
//	ExecutaComando(MDB_Comandos[58], UG.Comando.Remoto.Manual.VByPass.Fechar);
//	ExecutaComando(MDB_Comandos[59], UG.Comando.Remoto.Manual.Vborb.Abrir);
//	ExecutaComando(MDB_Comandos[60], UG.Comando.Remoto.Manual.Vborb.Fechar);
	ExecutaComando(MDB_Comandos[61], UG.Comando.Remoto.Manual.Comporta1.Abrir);
	ExecutaComando(MDB_Comandos[62], UG.Comando.Remoto.Manual.Comporta1.Fechar);
	ExecutaComando(MDB_Comandos[63], UG.Comando.Remoto.Manual.Comporta2.Abrir);
	ExecutaComando(MDB_Comandos[64], UG.Comando.Remoto.Manual.Comporta2.Fechar);
	ExecutaComando(MDB_Comandos[65], UG.Comando.Remoto.Manual.RV.Habilitar);
	ExecutaComando(MDB_Comandos[66], UG.Comando.Remoto.Manual.RV.Desabilitar);
	ExecutaComando(MDB_Comandos[67], UG.Comando.Remoto.Manual.RT.Habilitar);
	ExecutaComando(MDB_Comandos[68], UG.Comando.Remoto.Manual.RT.Desabilitar);
	ExecutaComando(MDB_Comandos[69], UG.Comando.Remoto.Manual.SC.Habilitar);
	ExecutaComando(MDB_Comandos[70], UG.Comando.Remoto.Manual.SC.Desabilitar);
//	ExecutaComando(MDB_Comandos[71], FALSE);
//	ExecutaComando(MDB_Comandos[72], FALSE);
//	ExecutaComando(MDB_Comandos[73], FALSE);
//	ExecutaComando(MDB_Comandos[74], FALSE);
//	ExecutaComando(MDB_Comandos[75], FALSE);
//	ExecutaComando(MDB_Comandos[76], FALSE);
//	ExecutaComando(MDB_Comandos[77], FALSE);
//	ExecutaComando(MDB_Comandos[78], FALSE);
//	ExecutaComando(MDB_Comandos[79], FALSE);
//	ExecutaComando(MDB_Comandos[80], FALSE);
	ExecutaComando(MDB_Comandos[81], Painel.Comando.Reset);
	ExecutaComando(MDB_Comandos[82], Painel.Comando.Cala_Sirene);
	ExecutaComando(MDB_Comandos[83], Painel.Comando.Emergencia.Ligar);
	ExecutaComando(MDB_Comandos[84], Painel.Comando.Emergencia.Desligar);
//	ExecutaComando(MDB_Comandos[85], FALSE);
//	ExecutaComando(MDB_Comandos[86], FALSE);
//	ExecutaComando(MDB_Comandos[87], FALSE);
//	ExecutaComando(MDB_Comandos[88], FALSE);
//	ExecutaComando(MDB_Comandos[89], FALSE);
//	ExecutaComando(MDB_Comandos[90], FALSE);
	ExecutaComando(MDB_Comandos[91], SFA.Comando.Bomba1.Ligar);
	ExecutaComando(MDB_Comandos[92], SFA.Comando.Bomba1.Desligar);
	ExecutaComando(MDB_Comandos[93], SFA.Comando.Bomba1.Reset_Horas);
	ExecutaComando(MDB_Comandos[94], SFA.Comando.Bomba1.Reset_Manobras);
//	ExecutaComando(MDB_Comandos[95], SFA.Comando.Retro_Lavagem);
	ExecutaComando(MDB_Comandos[96], SFA.Comando.Filtro1_Valv_Entrada1.Ligar);
	ExecutaComando(MDB_Comandos[97], SFA.Comando.Filtro1_Valv_Entrada1.Desligar);
	ExecutaComando(MDB_Comandos[98], SFA.Comando.Filtro1_Valv_Entrada2.Ligar);
	ExecutaComando(MDB_Comandos[99], SFA.Comando.Filtro1_Valv_Entrada2.Desligar);
	ExecutaComando(MDB_Comandos[100], SFA.Comando.Filtro1_Valv_Retrolav1.Ligar);
	ExecutaComando(MDB_Comandos[101], SFA.Comando.Filtro1_Valv_Retrolav1.Desligar);
	ExecutaComando(MDB_Comandos[102], SFA.Comando.Filtro1_Valv_Retrolav2.Ligar);
	ExecutaComando(MDB_Comandos[103], SFA.Comando.Filtro1_Valv_Retrolav2.Desligar);
	ExecutaComando(MDB_Comandos[104], SFA.Comando.Filtro2_Valv_Entrada1.Ligar);
	ExecutaComando(MDB_Comandos[105], SFA.Comando.Filtro2_Valv_Entrada1.Desligar);
	ExecutaComando(MDB_Comandos[106], SFA.Comando.Filtro2_Valv_Entrada2.Ligar);
	ExecutaComando(MDB_Comandos[107], SFA.Comando.Filtro2_Valv_Entrada2.Desligar);
	ExecutaComando(MDB_Comandos[108], SFA.Comando.Filtro2_Valv_Retrolav1.Ligar);
	ExecutaComando(MDB_Comandos[109], SFA.Comando.Filtro2_Valv_Retrolav1.Desligar);
	ExecutaComando(MDB_Comandos[110], SFA.Comando.Filtro2_Valv_Retrolav2.Ligar);
	ExecutaComando(MDB_Comandos[111], SFA.Comando.Filtro2_Valv_Retrolav2.Desligar);
//	ExecutaComando(MDB_Comandos[112], FALSE);
//	ExecutaComando(MDB_Comandos[113], FALSE);
//	ExecutaComando(MDB_Comandos[114], FALSE);
//	ExecutaComando(MDB_Comandos[115], FALSE);
//	ExecutaComando(MDB_Comandos[116], FALSE);
//	ExecutaComando(MDB_Comandos[117], FALSE);
//	ExecutaComando(MDB_Comandos[118], FALSE);
//	ExecutaComando(MDB_Comandos[119], FALSE);
//	ExecutaComando(MDB_Comandos[120], FALSE);
	ExecutaComando(MDB_Comandos[121], UHLM.Comando.Bomba1.Ligar);
	ExecutaComando(MDB_Comandos[122], UHLM.Comando.Bomba1.Desligar);
	ExecutaComando(MDB_Comandos[123], UHLM.Comando.Bomba1.Reset_Horas);
	ExecutaComando(MDB_Comandos[124], UHLM.Comando.Bomba1.Reset_Manobras);
	ExecutaComando(MDB_Comandos[125], UHLM.Comando.Bomba2.Ligar);
	ExecutaComando(MDB_Comandos[126], UHLM.Comando.Bomba2.Desligar);
	ExecutaComando(MDB_Comandos[127], UHLM.Comando.Bomba2.Reset_Horas);
	ExecutaComando(MDB_Comandos[128], UHLM.Comando.Bomba2.Reset_Manobras);
	ExecutaComando(MDB_Comandos[129], UHLM.Comando.JackingOil.Ligar);
	ExecutaComando(MDB_Comandos[130], UHLM.Comando.JackingOil.Desligar);
	ExecutaComando(MDB_Comandos[131], UHLM.Comando.JackingOil.Reset_Horas);
	ExecutaComando(MDB_Comandos[132], UHLM.Comando.JackingOil.Reset_Manobras);
	ExecutaComando(MDB_Comandos[133], UHLM.Comando.Ventilador.Ligar);
	ExecutaComando(MDB_Comandos[134], UHLM.Comando.Ventilador.Desligar);
	ExecutaComando(MDB_Comandos[135], UHLM.Comando.Ventilador.Reset_Horas);
	ExecutaComando(MDB_Comandos[136], UHLM.Comando.Ventilador.Reset_Manobras);
	ExecutaComando(MDB_Comandos[137], UHLM.Comando.Bomba3.Ligar);
	ExecutaComando(MDB_Comandos[138], UHLM.Comando.Bomba3.Desligar);
	ExecutaComando(MDB_Comandos[139], UHLM.Comando.Bomba3.Reset_Horas);
	ExecutaComando(MDB_Comandos[140], UHLM.Comando.Bomba3.Reset_Manobras);
//	ExecutaComando(MDB_Comandos[141], FALSE);
//	ExecutaComando(MDB_Comandos[142], FALSE);
//	ExecutaComando(MDB_Comandos[143], FALSE);
//	ExecutaComando(MDB_Comandos[144], FALSE);
//	ExecutaComando(MDB_Comandos[145], FALSE);
	ExecutaComando(MDB_Comandos[146], UHRV.Comando.Bomba1.Ligar);
	ExecutaComando(MDB_Comandos[147], UHRV.Comando.Bomba1.Desligar);
	ExecutaComando(MDB_Comandos[148], UHRV.Comando.Bomba1.Reset_Horas);
	ExecutaComando(MDB_Comandos[149], UHRV.Comando.Bomba1.Reset_Manobras);
	ExecutaComando(MDB_Comandos[150], UHRV.Comando.Bomba2.Ligar);
	ExecutaComando(MDB_Comandos[151], UHRV.Comando.Bomba2.Desligar);
	ExecutaComando(MDB_Comandos[152], UHRV.Comando.Bomba2.Reset_Horas);
	ExecutaComando(MDB_Comandos[153], UHRV.Comando.Bomba2.Reset_Manobras);
	ExecutaComando(MDB_Comandos[154], UHRV.Comando.Bomba3.Ligar);
	ExecutaComando(MDB_Comandos[155], UHRV.Comando.Bomba3.Desligar);
	ExecutaComando(MDB_Comandos[156], UHRV.Comando.Bomba3.Reset_Horas);
	ExecutaComando(MDB_Comandos[157], UHRV.Comando.Bomba3.Reset_Manobras);
	ExecutaComando(MDB_Comandos[158], UHRV.Comando.Vseg1.Ligar);
	ExecutaComando(MDB_Comandos[159], UHRV.Comando.Vseg1.Desligar);
	ExecutaComando(MDB_Comandos[160], UHRV.Comando.Vseg2.Ligar);
	ExecutaComando(MDB_Comandos[161], UHRV.Comando.Vseg2.Desligar);
	ExecutaComando(MDB_Comandos[162], UHRV.Comando.Ventagem.Ligar);
	ExecutaComando(MDB_Comandos[163], UHRV.Comando.Ventagem.Desligar);
//	ExecutaComando(MDB_Comandos[164], FALSE);
//	ExecutaComando(MDB_Comandos[165], FALSE);
//	ExecutaComando(MDB_Comandos[166], FALSE);
//	ExecutaComando(MDB_Comandos[167], FALSE);
//	ExecutaComando(MDB_Comandos[168], FALSE);
//	ExecutaComando(MDB_Comandos[169], FALSE);
//	ExecutaComando(MDB_Comandos[170], FALSE);
//	ExecutaComando(MDB_Comandos[171], FALSE);
//	ExecutaComando(MDB_Comandos[172], FALSE);
//	ExecutaComando(MDB_Comandos[173], FALSE);
//	ExecutaComando(MDB_Comandos[174], FALSE);
//	ExecutaComando(MDB_Comandos[175], FALSE);
//	ExecutaComando(MDB_Comandos[176], FALSE);
//	ExecutaComando(MDB_Comandos[177], FALSE);
//	ExecutaComando(MDB_Comandos[178], FALSE);
//	ExecutaComando(MDB_Comandos[179], FALSE);
//	ExecutaComando(MDB_Comandos[180], FALSE);
	ExecutaComando(MDB_Comandos[181], Freio.Comando.Modo_Continuo);
	ExecutaComando(MDB_Comandos[182], Freio.Comando.Modo_intermitente);
	ExecutaComando(MDB_Comandos[183], Freio.Comando.Aplicar);
	ExecutaComando(MDB_Comandos[184], Freio.Comando.Desaplicar);
//	ExecutaComando(MDB_Comandos[185], FALSE);
//	ExecutaComando(MDB_Comandos[186], FALSE);
//	ExecutaComando(MDB_Comandos[187], FALSE);
//	ExecutaComando(MDB_Comandos[188], FALSE);
//	ExecutaComando(MDB_Comandos[189], FALSE);
//	ExecutaComando(MDB_Comandos[190], FALSE);
//	ExecutaComando(MDB_Comandos[191], VByPass.Comando.VAbrir.Ligar);
//	ExecutaComando(MDB_Comandos[192], VByPass.Comando.VAbrir.Desligar);
//	ExecutaComando(MDB_Comandos[193], VByPass.Comando.VFechar.Ligar);
//	ExecutaComando(MDB_Comandos[194], VByPass.Comando.VFechar.Desligar);
//	ExecutaComando(MDB_Comandos[195], FALSE);
//	ExecutaComando(MDB_Comandos[196], FALSE);
//	ExecutaComando(MDB_Comandos[197], FALSE);
//	ExecutaComando(MDB_Comandos[198], FALSE);
//	ExecutaComando(MDB_Comandos[199], FALSE);
//	ExecutaComando(MDB_Comandos[200], FALSE);
//	ExecutaComando(MDB_Comandos[201], Vborb.Comando.VAbrir.Ligar);
//	ExecutaComando(MDB_Comandos[202], VBorb.Comando.VAbrir.Desligar);
//	ExecutaComando(MDB_Comandos[203], VBorb.Comando.VReter.Ligar);
//	ExecutaComando(MDB_Comandos[204], VBorb.Comando.VReter.Desligar);
//	ExecutaComando(MDB_Comandos[205], FALSE);
//	ExecutaComando(MDB_Comandos[206], FALSE);
//	ExecutaComando(MDB_Comandos[207], FALSE);
//	ExecutaComando(MDB_Comandos[208], FALSE);
//	ExecutaComando(MDB_Comandos[209], FALSE);
//	ExecutaComando(MDB_Comandos[210], FALSE);
	ExecutaComando(MDB_Comandos[211], Comporta1.Comando.Abertura.Ligar);
	ExecutaComando(MDB_Comandos[212], Comporta1.Comando.Abertura.Desligar);
	ExecutaComando(MDB_Comandos[213], Comporta1.Comando.Abertura_Lenta.Ligar);
	ExecutaComando(MDB_Comandos[214], Comporta1.Comando.Abertura_Lenta.Desligar);
	ExecutaComando(MDB_Comandos[215], Comporta1.Comando.Fechamento.Ligar);
	ExecutaComando(MDB_Comandos[216], Comporta1.Comando.Fechamento.Desligar);
	ExecutaComando(MDB_Comandos[217], Comporta1.Comando.Fechamento_Rapido.Ligar);
	ExecutaComando(MDB_Comandos[218], Comporta1.Comando.Fechamento_Rapido.Desligar);
	ExecutaComando(MDB_Comandos[219], Comporta_UH.Comando.Bomba1.Ligar);
	ExecutaComando(MDB_Comandos[220], Comporta_UH.Comando.Bomba1.Desligar);
	ExecutaComando(MDB_Comandos[221], Comporta_UH.Comando.Bomba1.Reset_Horas);
	ExecutaComando(MDB_Comandos[222], Comporta_UH.Comando.Bomba1.Reset_Manobras);
	ExecutaComando(MDB_Comandos[223], Comporta_UH.Comando.Bomba2.Ligar);
	ExecutaComando(MDB_Comandos[224], Comporta_UH.Comando.Bomba2.Desligar);
	ExecutaComando(MDB_Comandos[225], Comporta_UH.Comando.Bomba2.Reset_Horas);
	ExecutaComando(MDB_Comandos[226], Comporta_UH.Comando.Bomba2.Reset_Manobras);
//	ExecutaComando(MDB_Comandos[227], FALSE);
//	ExecutaComando(MDB_Comandos[228], FALSE);
//	ExecutaComando(MDB_Comandos[229], FALSE);
//	ExecutaComando(MDB_Comandos[230], FALSE);
//	ExecutaComando(MDB_Comandos[231], FALSE);
//	ExecutaComando(MDB_Comandos[232], FALSE);
//	ExecutaComando(MDB_Comandos[233], FALSE);
//	ExecutaComando(MDB_Comandos[234], FALSE);
//	ExecutaComando(MDB_Comandos[235], FALSE);
//	ExecutaComando(MDB_Comandos[236], FALSE);
//	ExecutaComando(MDB_Comandos[237], FALSE);
//	ExecutaComando(MDB_Comandos[238], FALSE);
//	ExecutaComando(MDB_Comandos[239], FALSE);
//	ExecutaComando(MDB_Comandos[240], FALSE);
	ExecutaComando(MDB_Comandos[241], RT.Comando.Qm_Constante);
	ExecutaComando(MDB_Comandos[242], RT.Comando.FP_Constante);
//	ExecutaComando(MDB_Comandos[243], FALSE);
//	ExecutaComando(MDB_Comandos[244], FALSE);
//	ExecutaComando(MDB_Comandos[245], FALSE);
//	ExecutaComando(MDB_Comandos[246], FALSE);
//	ExecutaComando(MDB_Comandos[247], FALSE);
//	ExecutaComando(MDB_Comandos[248], FALSE);
//	ExecutaComando(MDB_Comandos[249], FALSE);
//	ExecutaComando(MDB_Comandos[250], FALSE);
	ExecutaComando(MDB_Comandos[251], DJ52G.Comando.Abrir);
	ExecutaComando(MDB_Comandos[252], DJ52G.Comando.Carregar_Mola);
	ExecutaComando(MDB_Comandos[253], DJ52G.Comando.Bobina_Minima);
//	ExecutaComando(MDB_Comandos[254], FALSE);
//	ExecutaComando(MDB_Comandos[255], FALSE);
//	ExecutaComando(MDB_Comandos[256], FALSE);
//	ExecutaComando(MDB_Comandos[257], FALSE);
//	ExecutaComando(MDB_Comandos[258], FALSE);
//	ExecutaComando(MDB_Comandos[259], FALSE);
//	ExecutaComando(MDB_Comandos[260], FALSE);
//	ExecutaComando(MDB_Comandos[261], DJ52L.Comando.Abrir);
//	ExecutaComando(MDB_Comandos[262], DJ52L.Comando.Fechar);
//	ExecutaComando(MDB_Comandos[263], FALSE);
//	ExecutaComando(MDB_Comandos[264], FALSE);
//	ExecutaComando(MDB_Comandos[265], FALSE);
//	ExecutaComando(MDB_Comandos[266], FALSE);
//	ExecutaComando(MDB_Comandos[267], FALSE);
//	ExecutaComando(MDB_Comandos[268], FALSE);
//	ExecutaComando(MDB_Comandos[269], FALSE);
//	ExecutaComando(MDB_Comandos[270], FALSE);
	ExecutaComando(MDB_Comandos[271], Nivel.Comando.Habilitar);
	ExecutaComando(MDB_Comandos[272], Nivel.Comando.Desabilitar);
//	ExecutaComando(MDB_Comandos[273], FALSE);
//	ExecutaComando(MDB_Comandos[274], FALSE);
//	ExecutaComando(MDB_Comandos[275], FALSE);
//	ExecutaComando(MDB_Comandos[276], FALSE);
//	ExecutaComando(MDB_Comandos[277], FALSE);
//	ExecutaComando(MDB_Comandos[278], FALSE);
//	ExecutaComando(MDB_Comandos[279], FALSE);
//	ExecutaComando(MDB_Comandos[280], FALSE);

	//-------------------------------------------------------------------------------------------
END_PROGRAM
```

#### ExecutaComando.st
```iecst
(* TODO: Add your comment here *)
FUNCTION ExecutaComando
    IF in THEN
        in  := FALSE;
        out := TRUE;
    END_IF;
    ExecutaComando := TRUE;
END_FUNCTION
```

### Program Logical/Auto/Modbus/MDB_MED

#### Cyclic.st
```iecst
PROGRAM _CYCLIC
	//-------------------------------------------------------------------------------------------
	(*Medidas*)
	//-------------------------------------------------------------------------------------------

	MDB_Medidas[1] := UG.Medida.UP_Partindo_Tempo;
	MDB_Medidas[2] := UG.Medida.UPGM_Partindo_Tempo;
	MDB_Medidas[3] := UG.Medida.UMVD_Partindo_Tempo;
	MDB_Medidas[4] := UG.Medida.UPS_Partindo_Tempo;
	MDB_Medidas[5] := UG.Medida.US_Parando_Tempo;
	MDB_Medidas[6] := UG.Medida.UPS_Parando_Tempo;
	MDB_Medidas[7] := UG.Medida.UMVD_Parando_Tempo;
	MDB_Medidas[8] := UG.Medida.UPGM_Parando_Tempo;
	MDB_Medidas[9] := 0.0;
	MDB_Medidas[10] := 0.0;
	MDB_Medidas[11] := 0.0;
	MDB_Medidas[12] := 0.0;
	MDB_Medidas[13] := 0.0;
	MDB_Medidas[14] := 0.0;
	MDB_Medidas[15] := 0.0;
	MDB_Medidas[16] := 0.0;
	MDB_Medidas[17] := 0.0;
	MDB_Medidas[18] := 0.0;
	MDB_Medidas[19] := 0.0;
	MDB_Medidas[20] := 0.0;
	MDB_Medidas[21] := SFA.Medida.Bomba1.Numero_Manobras;
	MDB_Medidas[22] := SFA.Medida.Bomba1.Tempo_Giro;
	MDB_Medidas[23] := 0.0;
	MDB_Medidas[24] := 0.0;
	MDB_Medidas[25] := SFA.Medida.Pressao1_Lado_Limpo.Sensor;
	MDB_Medidas[26] := SFA.Medida.Pressao1_Lado_Limpo.Valor;
	MDB_Medidas[27] := SFA.Medida.Pressao2_Lado_Limpo.Sensor;
	MDB_Medidas[28] := SFA.Medida.Pressao2_Lado_Limpo.Valor;
	MDB_Medidas[29] := SFA.Medida.Pressao1_Lado_Sujo.Sensor;
	MDB_Medidas[30] := SFA.Medida.Pressao1_Lado_Sujo.Valor;
	MDB_Medidas[31] := SFA.Medida.Pressao2_Lado_Sujo.Sensor;
	MDB_Medidas[32] := SFA.Medida.Pressao2_Lado_Sujo.Valor;
	MDB_Medidas[33] := 0.0;
	MDB_Medidas[34] := 0.0;
	MDB_Medidas[35] := 0.0;
	MDB_Medidas[36] := 0.0;
	MDB_Medidas[37] := 0.0;
	MDB_Medidas[38] := 0.0;
	MDB_Medidas[39] := 0.0;
	MDB_Medidas[40] := 0.0;
	MDB_Medidas[41] := UHLM.Medida.Bomba1.Numero_Manobras;
	MDB_Medidas[42] := UHLM.Medida.Bomba1.Tempo_Giro;
	MDB_Medidas[43] := UHLM.Medida.Bomba2.Numero_Manobras;
	MDB_Medidas[44] := UHLM.Medida.Bomba2.Tempo_Giro;
	MDB_Medidas[45] := UHLM.Medida.JackingOil.Numero_Manobras;
	MDB_Medidas[46] := UHLM.Medida.JackingOil.Tempo_Giro;
	MDB_Medidas[47] := UHLM.Medida.Ventilador.Numero_Manobras;
	MDB_Medidas[48] := UHLM.Medida.Ventilador.Tempo_Giro;
	MDB_Medidas[49] := UHLM.Medida.Temperatura.Sensor;
	MDB_Medidas[50] := UHLM.Medida.Temperatura.Valor;
	MDB_Medidas[51] := UHLM.Medida.Vazao.Sensor;
	MDB_Medidas[52] := UHLM.Medida.Vazao.Valor;
	MDB_Medidas[53] := UHLM.Medida.Bomba3.Numero_Manobras;
	MDB_Medidas[54] := UHLM.Medida.Bomba3.Tempo_Giro;
	MDB_Medidas[55] := 0.0;
	MDB_Medidas[56] := 0.0;
	MDB_Medidas[57] := 0.0;
	MDB_Medidas[58] := 0.0;
	MDB_Medidas[59] := 0.0;
	MDB_Medidas[60] := 0.0;
	MDB_Medidas[61] := UHRV.Medida.Bomba1.Numero_Manobras;
	MDB_Medidas[62] := UHRV.Medida.Bomba1.Tempo_Giro;
	MDB_Medidas[63] := UHRV.Medida.Bomba2.Numero_Manobras;
	MDB_Medidas[64] := UHRV.Medida.Bomba2.Tempo_Giro;
	MDB_Medidas[65] := UHRV.Medida.Bomba3.Numero_Manobras;
	MDB_Medidas[66] := UHRV.Medida.Bomba3.Tempo_Giro;
	MDB_Medidas[67] := UHRV.Medida.Ventilador.Numero_Manobras;
	MDB_Medidas[68] := UHRV.Medida.Ventilador.Tempo_Giro;
	MDB_Medidas[69] := UHRV.Medida.Temperatura.Sensor;
	MDB_Medidas[70] := UHRV.Medida.Temperatura.Valor;
	MDB_Medidas[71] := UHRV.Medida.Pressao.Sensor;
	MDB_Medidas[72] := UHRV.Medida.Pressao.Valor;
	MDB_Medidas[73] := 0.0;
	MDB_Medidas[74] := 0.0;
	MDB_Medidas[75] := 0.0;
	MDB_Medidas[76] := 0.0;
	MDB_Medidas[77] := 0.0;
	MDB_Medidas[78] := 0.0;
	MDB_Medidas[79] := 0.0;
	MDB_Medidas[80] := 0.0;
//	MDB_Medidas[81] := VByPass.Medida.Tempo.Abrir;
//	MDB_Medidas[82] := VByPass.Medida.Tempo.Fechar;
	MDB_Medidas[83] := 0.0;
	MDB_Medidas[84] := 0.0;
	MDB_Medidas[85] := 0.0;
	MDB_Medidas[86] := 0.0;
	MDB_Medidas[87] := 0.0;
	MDB_Medidas[88] := 0.0;
	MDB_Medidas[89] := 0.0;
	MDB_Medidas[90] := 0.0;
//	MDB_Medidas[91] := Vborb.Medida.Tempo.Abrir;
//	MDB_Medidas[92] := Vborb.Medida.Tempo.Fechar;
//	MDB_Medidas[93] := Vborb.Medida.Tempo.Equalizar;
//	MDB_Medidas[94] := Vborb.Medida.Delta_Pressao;
//	MDB_Medidas[95] := Vborb.Medida.Pressao.Montante.Sensor;
//	MDB_Medidas[96] := Vborb.Medida.Pressao.Montante.Valor;
//	MDB_Medidas[97] := Vborb.Medida.Pressao.Jusante.Sensor;
//	MDB_Medidas[98] := Vborb.Medida.Pressao.Jusante.Valor;
	MDB_Medidas[99] := 0.0;
	MDB_Medidas[100] := 0.0;
	MDB_Medidas[101] := 0.0;
	MDB_Medidas[102] := 0.0;
	MDB_Medidas[103] := 0.0;
	MDB_Medidas[104] := 0.0;
	MDB_Medidas[105] := 0.0;
	MDB_Medidas[106] := 0.0;
	MDB_Medidas[107] := 0.0;
	MDB_Medidas[108] := 0.0;
	MDB_Medidas[109] := 0.0;
	MDB_Medidas[110] := 0.0;
	MDB_Medidas[111] := Comporta1.Medida.Tempo_Abertura;
	MDB_Medidas[112] := Comporta1.Medida.Tempo_Cracking;
	MDB_Medidas[113] := Comporta1.Medida.Tempo_Fechamento;
	MDB_Medidas[114] := Comporta1.Medida.Delta_Pressao;
	MDB_Medidas[115] := Comporta1.Medida.Encoder1_Sensor;
	MDB_Medidas[116] := Comporta1.Medida.Encoder1_Valor;
	MDB_Medidas[117] := Comporta2.Medida.Encoder2_Sensor;
	MDB_Medidas[118] := Comporta2.Medida.Encoder2_Valor;
	MDB_Medidas[119] := Comporta2.Medida.Tempo_Abertura;
	MDB_Medidas[120] := Comporta2.Medida.Tempo_Cracking;
	MDB_Medidas[121] := Comporta2.Medida.Tempo_Fechamento;
	MDB_Medidas[122] := Comporta2.Medida.Delta_Pressao;
	MDB_Medidas[123] := Comporta_UH.Medida.Temperatura_Oleo.Sensor;
	MDB_Medidas[124] := Comporta_UH.Medida.Temperatura_Oleo.Valor;
	MDB_Medidas[125] := Comporta_UH.Medida.Bomba1.Tempo_Giro;
	MDB_Medidas[126] := Comporta_UH.Medida.Bomba1.Numero_Manobras;
	MDB_Medidas[127] := Comporta_UH.Medida.Bomba2.Tempo_Giro;
	MDB_Medidas[128] := Comporta_UH.Medida.Bomba2.Numero_Manobras;
	MDB_Medidas[129] := 0.0;
	MDB_Medidas[130] := 0.0;
	MDB_Medidas[131] := Turbina.Medida.Gaxeteiro.Temperatura.Sensor;
	MDB_Medidas[132] := Turbina.Medida.Gaxeteiro.Temperatura.Valor;
	MDB_Medidas[133] := Turbina.Medida.Mancal1.Temperatura.Sensor;
	MDB_Medidas[134] := Turbina.Medida.Mancal1.Temperatura.Valor;
	MDB_Medidas[135] := Turbina.Medida.Mancal2.Temperatura.Sensor;
	MDB_Medidas[136] := Turbina.Medida.Mancal2.Temperatura.Valor;
	MDB_Medidas[137] := Turbina.Medida.Mancal3.Temperatura.Sensor;
	MDB_Medidas[138] := Turbina.Medida.Mancal3.Temperatura.Valor;
	MDB_Medidas[139] := Turbina.Medida.Mancal4.Temperatura.Sensor;
	MDB_Medidas[140] := Turbina.Medida.Mancal4.Temperatura.Valor;
	MDB_Medidas[141] := Turbina.Medida.Mancal5.Temperatura.Sensor;
	MDB_Medidas[142] := Turbina.Medida.Mancal5.Temperatura.Valor;
	MDB_Medidas[143] := Turbina.Medida.Mancal6.Temperatura.Sensor;
	MDB_Medidas[144] := Turbina.Medida.Mancal6.Temperatura.Valor;
	MDB_Medidas[145] := Turbina.Medida.CaixaEspiral.Pressao.Sensor;
	MDB_Medidas[146] := Turbina.Medida.CaixaEspiral.Pressao.Valor;
	MDB_Medidas[147] := 0.0;
	MDB_Medidas[148] := 0.0;
	MDB_Medidas[149] := 0.0;
	MDB_Medidas[150] := 0.0;
	MDB_Medidas[151] := 0.0;
	MDB_Medidas[152] := 0.0;
	MDB_Medidas[153] := 0.0;
	MDB_Medidas[154] := 0.0;
	MDB_Medidas[155] := 0.0;
	MDB_Medidas[156] := 0.0;
	MDB_Medidas[157] := 0.0;
	MDB_Medidas[158] := 0.0;
	MDB_Medidas[159] := 0.0;
	MDB_Medidas[160] := 0.0;
	MDB_Medidas[161] := Gerador.Medida.Fase_A.Temperatura.Sensor;
	MDB_Medidas[162] := Gerador.Medida.Fase_A.Temperatura.Valor;
	MDB_Medidas[163] := Gerador.Medida.Fase_B.Temperatura.Sensor;
	MDB_Medidas[164] := Gerador.Medida.Fase_B.Temperatura.Valor;
	MDB_Medidas[165] := Gerador.Medida.Fase_C.Temperatura.Sensor;
	MDB_Medidas[166] := Gerador.Medida.Fase_C.Temperatura.Valor;
	MDB_Medidas[167] := Gerador.Medida.NucleoEstatorico1.Temperatura.Sensor;
	MDB_Medidas[168] := Gerador.Medida.NucleoEstatorico1.Temperatura.Valor;
	MDB_Medidas[169] := Gerador.Medida.NucleoEstatorico2.Temperatura.Sensor;
	MDB_Medidas[170] := Gerador.Medida.NucleoEstatorico2.Temperatura.Valor;
	MDB_Medidas[171] := Gerador.Medida.NucleoEstatorico3.Temperatura.Sensor;
	MDB_Medidas[172] := Gerador.Medida.NucleoEstatorico3.Temperatura.Valor;
	MDB_Medidas[173] := Gerador.Medida.Mancal1.Temperatura.Sensor;
	MDB_Medidas[174] := Gerador.Medida.Mancal1.Temperatura.Valor;
	MDB_Medidas[175] := Gerador.Medida.Mancal2.Temperatura.Sensor;
	MDB_Medidas[176] := Gerador.Medida.Mancal2.Temperatura.Valor;
	MDB_Medidas[177] := Gerador.Medida.Mancal3.Temperatura.Sensor;
	MDB_Medidas[178] := Gerador.Medida.Mancal3.Temperatura.Valor;
	MDB_Medidas[179] := Gerador.Medida.Mancal4.Temperatura.Sensor;
	MDB_Medidas[180] := Gerador.Medida.Mancal4.Temperatura.Valor;
	MDB_Medidas[181] := Gerador.Medida.Mancal5.Temperatura.Sensor;
	MDB_Medidas[182] := Gerador.Medida.Mancal5.Temperatura.Valor;
	MDB_Medidas[183] := Gerador.Medida.Mancal6.Temperatura.Sensor;
	MDB_Medidas[184] := Gerador.Medida.Mancal6.Temperatura.Valor;
	MDB_Medidas[185] := 0.0;
	MDB_Medidas[186] := 0.0;
	MDB_Medidas[187] := 0.0;
	MDB_Medidas[188] := 0.0;
	MDB_Medidas[189] := 0.0;
	MDB_Medidas[190] := 0.0;
	MDB_Medidas[191] := 0.0;
	MDB_Medidas[192] := 0.0;
	MDB_Medidas[193] := 0.0;
	MDB_Medidas[194] := 0.0;
	MDB_Medidas[195] := 0.0;
	MDB_Medidas[196] := 0.0;
	MDB_Medidas[197] := 0.0;
	MDB_Medidas[198] := 0.0;
	MDB_Medidas[199] := 0.0;
	MDB_Medidas[200] := 0.0;
	MDB_Medidas[201] := Trafo_Exc.Medidas.Fase_A.Temperatura.Sensor;
	MDB_Medidas[202] := Trafo_Exc.Medidas.Fase_A.Temperatura.Valor;
	MDB_Medidas[203] := Trafo_Exc.Medidas.Fase_B.Temperatura.Sensor;
	MDB_Medidas[204] := Trafo_Exc.Medidas.Fase_B.Temperatura.Valor;
	MDB_Medidas[205] := Trafo_Exc.Medidas.Fase_C.Temperatura.Sensor;
	MDB_Medidas[206] := Trafo_Exc.Medidas.Fase_C.Temperatura.Valor;
	MDB_Medidas[207] := 0.0;
	MDB_Medidas[208] := 0.0;
	MDB_Medidas[209] := 0.0;
	MDB_Medidas[210] := 0.0;
	MDB_Medidas[211] := 0.0;
	MDB_Medidas[212] := 0.0;
	MDB_Medidas[213] := 0.0;
	MDB_Medidas[214] := 0.0;
	MDB_Medidas[215] := 0.0;
	MDB_Medidas[216] := 0.0;
	MDB_Medidas[217] := 0.0;
	MDB_Medidas[218] := 0.0;
	MDB_Medidas[219] := 0.0;
	MDB_Medidas[220] := 0.0;
	MDB_Medidas[221] := Nivel.Medida.Barragem.Valor;
	MDB_Medidas[222] := Nivel.Medida.Barragem.Sensor;
	MDB_Medidas[223] := Nivel.Medida.Jusante.Valor;
	MDB_Medidas[224] := Nivel.Medida.Jusante.Sensor;
	MDB_Medidas[225] := Nivel.Medida.Potencia;
	MDB_Medidas[226] := Nivel.Medida.Jusante_Grade1.Valor;
	MDB_Medidas[227] := Nivel.Medida.Jusante_Grade1.Sensor;
	MDB_Medidas[228] := Nivel.Medida.Jusante_Grade2.Valor;
	MDB_Medidas[229] := Nivel.Medida.Jusante_Grade2.Sensor;
	MDB_Medidas[230] := 0.0;

	//-------------------------------------------------------------------------------------------
END_PROGRAM
```

### Program Logical/Auto/Modbus/MDB_PAR
